			// code that is repeated every cycle in this state	
				IF iCurrentValveMode = 63 AND iCurrentChannelTM = 31 AND iCurrentTransferControlTM = 2 AND iCurrentAddressedTargetTM = usiChooseOtherValve AND iCurrentIndexTM = iCountMFLdownload + 50 THEN
					astMalfunctionlist[iCountMFLdownload].uiHours := WORD_TO_UINT(awBusDataFromVTEM[2]);				// Save hours
					
					xStateFinished := TRUE;
				END_IF
			//-----------------------------------------------------------------------------------------------------------
			
			// Transition
				IF xStateFinished = TRUE THEN
					xStateFinished := FALSE;
					xStateChange := TRUE;
					iState := 42;
					iCommandNumber := 42;
				END_IF
			//-----------------------------------------------------------------------------------------------------------
			
		42:	// READING MALFUNCTION MESSAGE TIME STAMP PART II
			// code that is executed only in the first cycle of this state
				IF xStateChange = TRUE THEN
					xStateChange := FALSE;
					iResponse := eResponseReadMalfunctionList.transferring;
					xDone := FALSE;
					xError := FALSE;
					xBusy := TRUE;
					xAborted := FALSE;
				END_IF
			//-----------------------------------------------------------------------------------------------------------

			// code that is repeated every cycle in this state	
				IF iCurrentValveMode = 63 AND iCurrentChannelTM = 31 AND iCurrentTransferControlTM = 2 AND iCurrentAddressedTargetTM = usiChooseOtherValve AND iCurrentIndexTM = iCountMFLdownload + 100 THEN
					fbreadbitsfromword(wData:=awBusDataFromVTEM[2], iStartBit:=8, iEndBit:=15, iValue:= , xError:=);		// Read minutes
					astMalfunctionlist[iCountMFLdownload].usiMinutes := INT_TO_USINT(fbreadbitsfromword.iValue);			// Save minutes
					
					fbreadbitsfromword(wData:=awBusDataFromVTEM[2], iStartBit:=0, iEndBit:=7, iValue:= , xError:=);			// Read seconds
					astMalfunctionlist[iCountMFLdownload].usiSeconds := INT_TO_USINT(fbreadbitsfromword.iValue);			// Save seconds
					
					xStateFinished := TRUE;
				END_IF
			//-----------------------------------------------------------------------------------------------------------
			
			// Transition
				IF xStateFinished = TRUE THEN
					xStateFinished := FALSE;
					xStateChange := TRUE;
					iState := 43;
					iCommandNumber := 43;
				END_IF
			//-----------------------------------------------------------------------------------------------------------

		43:	// READING MALFUNCTION MESSAGE TIME STAMP PART III
			// code that is executed only in the first cycle of this state
				IF xStateChange = TRUE THEN
					xStateChange := FALSE;
					iResponse := eResponseReadMalfunctionList.transferring;
					xDone := FALSE;
					xError := FALSE;
					xBusy := TRUE;
					xAborted := FALSE;
				END_IF
			//-----------------------------------------------------------------------------------------------------------
			
			// code that is repeated every cycle in this state	
				IF iCurrentValveMode = 63 AND iCurrentChannelTM = 31 AND iCurrentTransferControlTM = 2 AND iCurrentAddressedTargetTM = usiChooseOtherValve AND iCurrentIndexTM = iCountMFLdownload + 150 THEN
					astMalfunctionlist[iCountMFLdownload].uiMilliseconds := WORD_TO_UINT(awBusDataFromVTEM[2]);			// Save milliseconds
					
					IF iCountMFLdownload = iNumberOfMalfunctions THEN
						xReadProcessFinished := TRUE;
					ELSE
						xReadProcessFinished := FALSE;
						xStateFinished := TRUE;
					END_IF
				END_IF
			//-----------------------------------------------------------------------------------------------------------
			
			// Transition
				IF xReadProcessFinished = TRUE THEN
					xStateChange := TRUE;
					xStateFinished := FALSE;
					iState := 44;
					iCommandNumber := 44;
				ELSIF xStateFinished = TRUE THEN
					xStateFinished := FALSE;
					xStateChange := TRUE;
					iState := 40;
					iCountMFLdownload := iCountMFLdownload + 1;
					iCommandNumber := 40;
				END_IF
			//-----------------------------------------------------------------------------------------------------------
			
		44:	// READING TIME CODE OF MALFUNCTION LIST PART I
			// code that is executed only in the first cycle of this state
				IF xStateChange = TRUE THEN
					xStateChange := FALSE;
					iResponse := eResponseReadMalfunctionList.transferring;
					xDone := FALSE;
					xError := FALSE;
					xBusy := TRUE;
					xAborted := FALSE;
				END_IF
			//-----------------------------------------------------------------------------------------------------------
			
			// code that is repeated every cycle in this state	
				IF iCurrentValveMode = 63 AND iCurrentChannelTM = 31 AND iCurrentTransferControlTM = 2 AND iCurrentAddressedTargetTM = usiChooseOtherValve AND iCurrentIndexTM = 250 THEN
					stTimeStampList.uiHours := WORD_TO_UINT(awBusDataFromVTEM[2]);											// Save Hours
					
					xStateFinished := TRUE;
				END_IF
			//-----------------------------------------------------------------------------------------------------------
			
			// Transition
				IF xStateFinished = TRUE THEN
					xStateFinished := FALSE;
					xStateChange := TRUE;
					iState := 45;
					iCommandNumber := 45;
				END_IF
			//-----------------------------------------------------------------------------------------------------------
		
		45:	// READING TIME CODE OF MALFUNCTION LIST PART III
			// code that is executed only in the first cycle of this state
				IF xStateChange = TRUE THEN
					xStateChange := FALSE;
					iResponse := eResponseReadMalfunctionList.transferring;
					xDone := FALSE;
					xError := FALSE;
					xBusy := TRUE;
					xAborted := FALSE;
				END_IF
			//-----------------------------------------------------------------------------------------------------------
			
			// code that is repeated every cycle in this state	
				IF iCurrentValveMode = 63 AND iCurrentChannelTM = 31 AND iCurrentTransferControlTM = 2 AND iCurrentAddressedTargetTM = usiChooseOtherValve AND iCurrentIndexTM = 251 THEN
					fbreadbitsfromword(wData:=awBusDataFromVTEM[2], iStartBit:=8, iEndBit:=15, iValue:= , xError:=);		// Read minutes
					stTimeStampList.usiMinutes := INT_TO_USINT(fbreadbitsfromword.iValue);									// Save minutes

					fbreadbitsfromword(wData:=awBusDataFromVTEM[2], iStartBit:=0, iEndBit:=7, iValue:= , xError:=);			// Read seconds
					stTimeStampList.usiSeconds := INT_TO_USINT(fbreadbitsfromword.iValue);									// Save seconds
					
					xStateFinished := TRUE;
				END_IF
			//-----------------------------------------------------------------------------------------------------------
			
			// Transition
				IF xStateFinished = TRUE THEN
					xStateFinished := FALSE;
					xStateChange := TRUE;
					iState := 46;
					iCommandNumber := 46;
				END_IF
			//-----------------------------------------------------------------------------------------------------------
		
		46:	// READING TIME CODE OF MALFUNCTION LIST PART III
			// code that is executed only in the first cycle of this state
				IF xStateChange = TRUE THEN
					xStateChange := FALSE;
					iResponse := eResponseReadMalfunctionList.transferring;
					xDone := FALSE;
					xError := FALSE;
					xBusy := TRUE;
					xAborted := FALSE;
				END_IF
			//-----------------------------------------------------------------------------------------------------------
			
			// code that is repeated every cycle in this state	
				IF iCurrentValveMode = 63 AND iCurrentChannelTM = 31 AND iCurrentTransferControlTM = 2 AND iCurrentAddressedTargetTM = usiChooseOtherValve AND iCurrentIndexTM = 252 THEN
					stTimeStampList.uiMilliseconds := WORD_TO_UINT(awBusDataFromVTEM[2]);									// Save milliseconds
					
					xStateFinished := TRUE;
				END_IF
			//-----------------------------------------------------------------------------------------------------------
			
			// Transition
				IF xStateFinished = TRUE THEN
					xStateFinished := FALSE;
					xStateChange := TRUE;
					iState := 50;
				END_IF
			//-----------------------------------------------------------------------------------------------------------
		
		50:	// DONE
			// code that is executed only in the first cycle of this state
				IF xStateChange = TRUE THEN
					xStateChange := FALSE;
					iResponse := eResponseReadMalfunctionList.done;
					xDone := TRUE;
					xError := FALSE;
					xBusy := FALSE;
					xAborted := FALSE;
				END_IF
			//-----------------------------------------------------------------------------------------------------------
			
			// code that is repeated every cycle in this state	
				iCommandNumber := 5;	// exit transfer mode
			//-----------------------------------------------------------------------------------------------------------
			
			// Transition
				IF xExecute = FALSE THEN
					xStateChange := TRUE;
					iState := 100;
				END_IF
			//-----------------------------------------------------------------------------------------------------------
			
		51:	// DONE WITH EMPTY MALFUNCTION LIST
			// code that is executed only in the first cycle of this state
				IF xStateChange = TRUE THEN
					xStateChange := FALSE;
					iResponse := eResponseReadMalfunctionList.no_entries_in_malfunction_list;
					xDone := TRUE;
					xError := FALSE;
					xBusy := FALSE;
					xAborted := FALSE;
				END_IF
			//-----------------------------------------------------------------------------------------------------------
			
			// code that is repeated every cycle in this state	
				iCommandNumber := 5;	// exit transfer mode
			//-----------------------------------------------------------------------------------------------------------
			
			// Transition
				IF xExecute = FALSE THEN
					xStateChange := TRUE;
					iState := 100;
				END_IF
			//-----------------------------------------------------------------------------------------------------------
			
		70:	// ERROR
			// code that is executed only in the first cycle of this state
				IF xStateChange = TRUE THEN
					xStateChange := FALSE;
					iResponse := eResponseReadMalfunctionList.error_while_transmitting_data_to_vtem;
					xDone := FALSE;
					xError := TRUE;
					xBusy := FALSE;
					xAborted := FALSE;
				END_IF
			//-----------------------------------------------------------------------------------------------------------
				IF xInputConsistent = FALSE THEN
					iResponse := eResponseReadMalfunctionList.FB_needs_rising_edge_xExecute;
				END_IF
			
			// code that is repeated every cycle in this state	
				CASE iCurrentAppState OF
					1:	iResponse := eResponseReadMalfunctionList.invalid_SetValveMode;
					2:	iResponse := eResponseReadMalfunctionList.invalid_SetAppControl;
					3:	iResponse := eResponseReadMalfunctionList.invalid_SetAppOption;
					4:	iResponse := eResponseReadMalfunctionList.invalid_SetPointValue1;
					5:	iResponse := eResponseReadMalfunctionList.invalid_SetPointValue2;
					6:	iResponse := eResponseReadMalfunctionList.invalid_configuration;
					
					10:	iResponse := eResponseReadMalfunctionList.access_denied_WebConfig;
					11:	iResponse := eResponseReadMalfunctionList.access_denied_saving_parameterisation;
					12:	iResponse := eResponseReadMalfunctionList.no_license_for_this_MA;
					13:	iResponse := eResponseReadMalfunctionList.all_licenses_in_use;
					14:	iResponse := eResponseReadMalfunctionList.invalid_license_file;
					15:	iResponse := eResponseReadMalfunctionList.no_valve_detected;
					16:	iResponse := eResponseReadMalfunctionList.valve_self_calibration_running;
				END_CASE
			//-----------------------------------------------------------------------------------------------------------
			
			// Transition
				IF xExecute = FALSE AND xAbort = FALSE THEN
					xStateChange := TRUE;
					iState := 100;
				END_IF
			//-----------------------------------------------------------------------------------------------------------
			
		71:	// ERROR DURING TRANFER MODE
			// code that is executed only in the first cycle of this state
				IF xStateChange = TRUE THEN
					xStateChange := FALSE;
					xDone := FALSE;
					xError := TRUE;
					xBusy := FALSE;
					xAborted := FALSE;
				END_IF
			//-----------------------------------------------------------------------------------------------------------
			
			// code that is repeated every cycle in this state	
				CASE iCurrentValueTM OF
					1:	iResponse := eResponseReadMalfunctionList.invalid_Channel;
					2:	iResponse := eResponseReadMalfunctionList.invalid_TransferControl;
					3:	iResponse := eResponseReadMalfunctionList.invalid_usiChooseOtherValve; // invalid_AddtessedTarget is always invalid_usiChooseOtherValve
					4:	iResponse := eResponseReadMalfunctionList.invalid_Index;
					5:	iResponse := eResponseReadMalfunctionList.invalid_TransferValue;
					6:	iResponse := eResponseReadMalfunctionList.no_data_empty_slot;	// invalid_Combination is always no_data_empty_slot in the context of this function block
					7:	iResponse := eResponseReadMalfunctionList.access_denied_DataInUse;
					8:	iResponse := eResponseReadMalfunctionList.no_data_empty_slot;
				END_CASE
			//-----------------------------------------------------------------------------------------------------------
			
			// Transition
				IF xExecute = FALSE AND xAbort = FALSE THEN
					xStateChange := TRUE;
					iState := 100;
				END_IF
			//-----------------------------------------------------------------------------------------------------------
			
		80:	// ABORTING
			// code that is executed only in the first cycle of this state
				IF xStateChange = TRUE THEN
					xStateChange := FALSE;
					iResponse := eResponseReadMalfunctionList.aborting;
					xBusy := FALSE;
					xDone := FALSE;
					xError := FALSE;
					xAborted := TRUE;
				END_IF
			//-----------------------------------------------------------------------------------------------------------
			
			// code that is repeated every cycle in this state
				IF iCurrentValveMode = 63 THEN
					iCommandNumber := 5;	// exit transfer mode
				ELSIF iCurrentValveMode <> 61 AND iCurrentValveMode <> 63 THEN
					iCommandNumber := 6;	// stop running motion apps
				ELSE
					iCommandNumber := 0; 
				END_IF
			//-----------------------------------------------------------------------------------------------------------
			
			// Transition
				IF xAbort = FALSE AND xExecute = FALSE AND iCurrentValveMode = 61 THEN
					xStateChange := TRUE;
					iState := 100;
				END_IF
			//-----------------------------------------------------------------------------------------------------------

		100:	// RESETTING FUNCTION BLOCK AND VALVE
			// code that is executed only in the first cycle of this state
				IF xStateChange = TRUE THEN
					xStateChange := FALSE;
					iResponse := eResponseReadMalfunctionList.resetting;
					xDone := FALSE;
					xError := FALSE;
					xBusy := FALSE;
					xAborted := FALSE;
					xFirstTransfer := FALSE;
				END_IF
			//-----------------------------------------------------------------------------------------------------------
			
			// code that is repeated every cycle in this state	
				IF iCurrentValveMode = 63 THEN
					iCommandNumber := 5;	// exit transfer mode
				ELSIF iCurrentValveMode <> 61 AND iCurrentValveMode <> 63 THEN
					iCommandNumber := 6;	// stop running motion apps
				END_IF
				
				FOR iCountMFLreset := 1 TO 40 BY 1 DO
					astMalfunctionlist[iCountMFLreset].usiMalfunctionCode := 0;
					astMalfunctionlist[iCountMFLreset].usiMalfunctionSubcode := 0;
					astMalfunctionlist[iCountMFLreset].usiMalfunctionClassification := 0;
					astMalfunctionlist[iCountMFLreset].uiHours := 0;
					astMalfunctionlist[iCountMFLreset].usiMinutes := 0;
					astMalfunctionlist[iCountMFLreset].usiSeconds := 0;
					astMalfunctionlist[iCountMFLreset].uiMilliseconds := 0;
				END_FOR
				
				stTimeStampList.uiHours := 0;
				stTimeStampList.usiMinutes := 0;
				stTimeStampList.usiSeconds := 0;
				stTimeStampList.uiMilliseconds := 0;
				
				iNumberOfMalfunctions := 0;
				
				iCountMFLreset := 0;
				iCountMFLdownload := 1;
				xReadProcessFinished := FALSE;
				xStateFinished := FALSE;
			//-----------------------------------------------------------------------------------------------------------
			
			// Transition
				IF iCurrentValveMode = 61 THEN
					iCommandNumber := 6; // Last command to send before the FB is in IDLE
					xStateChange := TRUE;
					iState := 10;
				END_IF
			//-----------------------------------------------------------------------------------------------------------
			
	END_CASE
//-----------------------------------------------------------------------------------------------------------

// command section
	CASE iCommandNumber OF
		0:	// IDLE
			;
		
		5:	// EXIT TRANSFER MODE
			fbwritevaluetoword(iValue:=63, iStartBit:=0, iEndBit:=5, wDataWord:=awBusDataToVTEM[0], xError=> );							// Valve Mode = 63
			fbwritevaluetoword(iValue:=0, iStartBit:=6, iEndBit:=7, wDataWord:=awBusDataToVTEM[0], xError=> );							// 0 (unused)
			fbwritevaluetoword(iValue:=0, iStartBit:=8, iEndBit:=12, wDataWord:=awBusDataToVTEM[0], xError=> );							// Channel = 0 (ignored)
			fbwritevaluetoword(iValue:=3, iStartBit:=13, iEndBit:=15, wDataWord:=awBusDataToVTEM[0], xError=> );						// Transfer Control = Exit transfer mode (3)
			fbwritevaluetoword(iValue:=0, iStartBit:=0, iEndBit:=7, wDataWord:=awBusDataToVTEM[1], xError=> );							// Addressed Target = 0 (ignored)
			fbwritevaluetoword(iValue:=0, iStartBit:=8, iEndBit:=15, wDataWord:=awBusDataToVTEM[1], xError=> );							// Index = 0 (ignored)
			fbwritevaluetoword(iValue:=0, iStartBit:=0, iEndBit:=15, wDataWord:=awBusDataToVTEM[2], xError=> );							// Value = 0 (ignored)
			
		6:	// stop running motion apps
			fbwritevaluetoword(iValue:=61, iStartBit:=0, iEndBit:=5, wDataWord:=awBusDataToVTEM[0], xError=> );							// Valve Mode = 61 (stop)
			fbwritevaluetoword(iValue:=0, iStartBit:=6, iEndBit:=7, wDataWord:=awBusDataToVTEM[0], xError=> );							// App Control = 0 (unused)
			fbwritevaluetoword(iValue:=0, iStartBit:=8, iEndBit:=15, wDataWord:=awBusDataToVTEM[0], xError=> );							// App Option = 0 (unused)
			fbwritevaluetoword(iValue:=0, iStartBit:=0, iEndBit:=15, wDataWord:=awBusDataToVTEM[1], xError=> );							// Setpoint Value 1 = 0 (unused)
			fbwritevaluetoword(iValue:=0, iStartBit:=0, iEndBit:=15, wDataWord:=awBusDataToVTEM[2], xError=> );							// Setpoint Value 2 = 0 (unused)
		
		10:	// getting count of malfunction messages
			fbwritevaluetoword(iValue:=63, iStartBit:=0, iEndBit:=5, wDataWord:=awBusDataToVTEM[0], xError=> );							// Valve Mode = 63 (transfer mode)
			fbwritevaluetoword(iValue:=0, iStartBit:=6, iEndBit:=7, wDataWord:=awBusDataToVTEM[0], xError=> );							// 0 (unused)
			fbwritevaluetoword(iValue:=31, iStartBit:=8, iEndBit:=12, wDataWord:=awBusDataToVTEM[0], xError=> );						// Channel = 31 (malfunctions)
			fbwritevaluetoword(iValue:=2, iStartBit:=13, iEndBit:=15, wDataWord:=awBusDataToVTEM[0], xError=> );						// Transfer Control = 2 (Upload)
			fbwritevaluetoword(iValue:=usiChooseOtherValve, iStartBit:=0, iEndBit:=7, wDataWord:=awBusDataToVTEM[1], xError=> );		// Addressed Target = usiChooseOtherValve
			fbwritevaluetoword(iValue:=255, iStartBit:=8, iEndBit:=15, wDataWord:=awBusDataToVTEM[1], xError=> );						// Index = 255 (Number of malfunction messages)
			fbwritevaluetoword(iValue:=0, iStartBit:=0, iEndBit:=15, wDataWord:=awBusDataToVTEM[2], xError=> );							// Value = 0 (Upload)
		
		40:	// reading malfunction list
			fbwritevaluetoword(iValue:=63, iStartBit:=0, iEndBit:=5, wDataWord:=awBusDataToVTEM[0], xError=> );							// Valve Mode = 63 (transfer mode)
			fbwritevaluetoword(iValue:=0, iStartBit:=6, iEndBit:=7, wDataWord:=awBusDataToVTEM[0], xError=> );							// 0 (unused)
			fbwritevaluetoword(iValue:=31, iStartBit:=8, iEndBit:=12, wDataWord:=awBusDataToVTEM[0], xError=> );						// Channel = 31 (malfunctions)
			fbwritevaluetoword(iValue:=2, iStartBit:=13, iEndBit:=15, wDataWord:=awBusDataToVTEM[0], xError=> );						// Transfer Control = 2 (Upload)
			fbwritevaluetoword(iValue:=usiChooseOtherValve, iStartBit:=0, iEndBit:=7, wDataWord:=awBusDataToVTEM[1], xError=> );		// Addressed Target = usiChooseOtherValve
			fbwritevaluetoword(iValue:=iCountMFLdownload, iStartBit:=8, iEndBit:=15, wDataWord:=awBusDataToVTEM[1], xError=> );			// Index = iCounterMFLdownload (malfunction message)
			fbwritevaluetoword(iValue:=0, iStartBit:=0, iEndBit:=15, wDataWord:=awBusDataToVTEM[2], xError=> );							// Value = 0 (Upload)

		41:	// reading malfunction entry time stamp part I
			fbwritevaluetoword(iValue:=63, iStartBit:=0, iEndBit:=5, wDataWord:=awBusDataToVTEM[0], xError=> );							// Valve Mode = 63 (transfer mode)
			fbwritevaluetoword(iValue:=0, iStartBit:=6, iEndBit:=7, wDataWord:=awBusDataToVTEM[0], xError=> );							// 0 (unused)
			fbwritevaluetoword(iValue:=31, iStartBit:=8, iEndBit:=12, wDataWord:=awBusDataToVTEM[0], xError=> );						// Channel = 31 (malfunctions)
			fbwritevaluetoword(iValue:=2, iStartBit:=13, iEndBit:=15, wDataWord:=awBusDataToVTEM[0], xError=> );						// Transfer Control = 2 (Upload)
			fbwritevaluetoword(iValue:=usiChooseOtherValve, iStartBit:=0, iEndBit:=7, wDataWord:=awBusDataToVTEM[1], xError=> );		// Addressed Target = usiChooseOtherValve
			fbwritevaluetoword(iValue:=iCountMFLdownload+50, iStartBit:=8, iEndBit:=15, wDataWord:=awBusDataToVTEM[1], xError=> );		// Index = iCounterMFLdownload + 50 (time stamp of malfunction message, part I)
			fbwritevaluetoword(iValue:=0, iStartBit:=0, iEndBit:=15, wDataWord:=awBusDataToVTEM[2], xError=> );							// Value = 0 (Upload)
			
		42:	// reading malfunction entry time stamp part II
			fbwritevaluetoword(iValue:=63, iStartBit:=0, iEndBit:=5, wDataWord:=awBusDataToVTEM[0], xError=> );							// Valve Mode = 63 (transfer mode)
			fbwritevaluetoword(iValue:=0, iStartBit:=6, iEndBit:=7, wDataWord:=awBusDataToVTEM[0], xError=> );							// 0 (unused)
			fbwritevaluetoword(iValue:=31, iStartBit:=8, iEndBit:=12, wDataWord:=awBusDataToVTEM[0], xError=> );						// Channel = 31 (malfunctions)
			fbwritevaluetoword(iValue:=2, iStartBit:=13, iEndBit:=15, wDataWord:=awBusDataToVTEM[0], xError=> );						// Transfer Control = 2 (Upload)
			fbwritevaluetoword(iValue:=usiChooseOtherValve, iStartBit:=0, iEndBit:=7, wDataWord:=awBusDataToVTEM[1], xError=> );		// Addressed Target = usiChooseOtherValve
			fbwritevaluetoword(iValue:=iCountMFLdownload+100, iStartBit:=8, iEndBit:=15, wDataWord:=awBusDataToVTEM[1], xError=> );		// Index = iCounterMFLdownload + 100 (time stamp of malfunction message, part II)
			fbwritevaluetoword(iValue:=0, iStartBit:=0, iEndBit:=15, wDataWord:=awBusDataToVTEM[2], xError=> );							// Value = 0 (Upload)

		43: // reading malfunction entry time stamp part III
			fbwritevaluetoword(iValue:=63, iStartBit:=0, iEndBit:=5, wDataWord:=awBusDataToVTEM[0], xError=> );							// Valve Mode = 63 (transfer mode)
			fbwritevaluetoword(iValue:=0, iStartBit:=6, iEndBit:=7, wDataWord:=awBusDataToVTEM[0], xError=> );							// 0 (unused)
			fbwritevaluetoword(iValue:=31, iStartBit:=8, iEndBit:=12, wDataWord:=awBusDataToVTEM[0], xError=> );						// Channel = 31 (malfunctions)
			fbwritevaluetoword(iValue:=2, iStartBit:=13, iEndBit:=15, wDataWord:=awBusDataToVTEM[0], xError=> );						// Transfer Control = 2 (Upload)
			fbwritevaluetoword(iValue:=usiChooseOtherValve, iStartBit:=0, iEndBit:=7, wDataWord:=awBusDataToVTEM[1], xError=> );		// Addressed Target = usiChooseOtherValve
			fbwritevaluetoword(iValue:=iCountMFLdownload+150, iStartBit:=8, iEndBit:=15, wDataWord:=awBusDataToVTEM[1], xError=> );		// Index = iCounterMFLdownload + 150 (time stamp of malfunction message, part III)
			fbwritevaluetoword(iValue:=0, iStartBit:=0, iEndBit:=15, wDataWord:=awBusDataToVTEM[2], xError=> );							// Value = 0 (Upload)
		
		44:	// reading time stamp of malfunction list part I
			fbwritevaluetoword(iValue:=63, iStartBit:=0, iEndBit:=5, wDataWord:=awBusDataToVTEM[0], xError=> );							// Valve Mode = 63 (transfer mode)
			fbwritevaluetoword(iValue:=0, iStartBit:=6, iEndBit:=7, wDataWord:=awBusDataToVTEM[0], xError=> );							// 0 (unused)
			fbwritevaluetoword(iValue:=31, iStartBit:=8, iEndBit:=12, wDataWord:=awBusDataToVTEM[0], xError=> );						// Channel = 31 (malfunctions)
			fbwritevaluetoword(iValue:=2, iStartBit:=13, iEndBit:=15, wDataWord:=awBusDataToVTEM[0], xError=> );						// Transfer Control = 2 (Upload)
			fbwritevaluetoword(iValue:=usiChooseOtherValve, iStartBit:=0, iEndBit:=7, wDataWord:=awBusDataToVTEM[1], xError=> );		// Addressed Target = usiChooseOtherValve
			fbwritevaluetoword(iValue:=250, iStartBit:=8, iEndBit:=15, wDataWord:=awBusDataToVTEM[1], xError=> );						// Index = 250 (time stamp of malfunction list, part I)
			fbwritevaluetoword(iValue:=0, iStartBit:=0, iEndBit:=15, wDataWord:=awBusDataToVTEM[2], xError=> );							// Value = 0 (Upload)
		
		45:	// reading time stamp of malfunction list part II
			fbwritevaluetoword(iValue:=63, iStartBit:=0, iEndBit:=5, wDataWord:=awBusDataToVTEM[0], xError=> );							// Valve Mode = 63 (transfer mode)
			fbwritevaluetoword(iValue:=0, iStartBit:=6, iEndBit:=7, wDataWord:=awBusDataToVTEM[0], xError=> );							// 0 (unused)
			fbwritevaluetoword(iValue:=31, iStartBit:=8, iEndBit:=12, wDataWord:=awBusDataToVTEM[0], xError=> );						// Channel = 31 (malfunctions)
			fbwritevaluetoword(iValue:=2, iStartBit:=13, iEndBit:=15, wDataWord:=awBusDataToVTEM[0], xError=> );						// Transfer Control = 2 (Upload)
			fbwritevaluetoword(iValue:=usiChooseOtherValve, iStartBit:=0, iEndBit:=7, wDataWord:=awBusDataToVTEM[1], xError=> );		// Addressed Target = usiChooseOtherValve
			fbwritevaluetoword(iValue:=251, iStartBit:=8, iEndBit:=15, wDataWord:=awBusDataToVTEM[1], xError=> );						// Index = 251 (time stamp of malfunction list, part II)
			fbwritevaluetoword(iValue:=0, iStartBit:=0, iEndBit:=15, wDataWord:=awBusDataToVTEM[2], xError=> );							// Value = 0 (Upload)
		
		46:	// reading time stamp of malfunction list part III
			fbwritevaluetoword(iValue:=63, iStartBit:=0, iEndBit:=5, wDataWord:=awBusDataToVTEM[0], xError=> );							// Valve Mode = 63 (transfer mode)
			fbwritevaluetoword(iValue:=0, iStartBit:=6, iEndBit:=7, wDataWord:=awBusDataToVTEM[0], xError=> );							// 0 (unused)
			fbwritevaluetoword(iValue:=31, iStartBit:=8, iEndBit:=12, wDataWord:=awBusDataToVTEM[0], xError=> );						// Channel = 31 (malfunctions)
			fbwritevaluetoword(iValue:=2, iStartBit:=13, iEndBit:=15, wDataWord:=awBusDataToVTEM[0], xError=> );						// Transfer Control = 2 (Upload)
			fbwritevaluetoword(iValue:=usiChooseOtherValve, iStartBit:=0, iEndBit:=7, wDataWord:=awBusDataToVTEM[1], xError=> );		// Addressed Target = usiChooseOtherValve
			fbwritevaluetoword(iValue:=252, iStartBit:=8, iEndBit:=15, wDataWord:=awBusDataToVTEM[1], xError=> );						// Index = 252 (time stamp of malfunction list, part III)
			fbwritevaluetoword(iValue:=0, iStartBit:=0, iEndBit:=15, wDataWord:=awBusDataToVTEM[2], xError=> );							// Value = 0 (Upload)

	END_CASE	
//-----------------------------------------------------------------------------------------------------------

END_FUNCTION_BLOCK

// Transfermode/specific_MA_config/FB_Write_config_MA_10
// This function block can be used to download the configuration of Motion App 10 ("Flow control").
// The specific parameters of this Motion App are the inputs of this FB and can be defined by the user. 
// The function block uses the transfer mode to write this configuration to the Motion Terminal
// and indicates the state of the download process.

FUNCTION_BLOCK FB_Write_config_MA_10
VAR_INPUT
	awBusDataFromVTEM 				: ARRAY [0..2] OF WORD;		(* 6 bytes of process data received from the Motion Terminal *)
END_VAR
	
VAR_IN_OUT
	awBusDataToVTEM 				: ARRAY [0..2] OF WORD; 	(* 6 bytes of process data sent to the Motion Terminal *)
END_VAR

VAR_INPUT
	xExecute 						: BOOL; 					(* has to be set to TRUE for a download and to FALSE to reset the function block after a download *)

	iParameterSet					: INT := 1; 				(* the parameter set to be written to, 1 by default *)
	
	// system parameters
		iOperatingMedium			: eMA10OperatingMedium := 1;// Type and condition of the operating medium (values see eMA10OperatingMedium)
		iInPortFlowRate2_optional	: INT;						// Sensor port for flow rate at (2) (required for closed-loop controlled operating mode, value is number of the slot (beginning from 0 and including valve slots) * 10 + number of the port 
		iInPortFlowRate4_optional	: INT;						// Sensor port for flow rate at (4) (required for closed-loop controlled operating mode, value is number of the slot (beginning from 0 and including valve slots) * 10 + number of the port
		iInPortRetracted_optional	: INT;						// Sensor port for detection of end position at pressurisation of outlet port 2 (retracted), value is number of the slot (beginning from 0 and including valve slots) * 10 + number of the port
		iInPortAdvanced_optional	: INT;						// Sensor port for detection of end position at pressurisation of outlet port 4 (advanced), value is number of the slot (beginning from 0 and including valve slots) * 10 + number of the port

	// application parameters
		iCharacteristicAt2			: INT;						// Control characteristic, outlet port (2) (0 = "fast" (short tubes), 1 = medium (medium length tubes), 2 = "universal" (esp. long tubes), 3 = defined by tuning parameters (only if closed-loop control is activated for outlet port (2)))
		iCharacteristicAt4			: INT;						// Control characteristic, outlet port (4) (0 = "fast" (short tubes), 1 = medium (medium length tubes), 2 = "universal" (esp. long tubes), 3 = defined by tuning parameters (only if closed-loop control is activated for outlet port (4)))
		xClosedLoopControl2			: BOOL := FALSE;			// TRUE acivates closed-loop control for outlet port (2), FALSE is open-loop controlled operation
		xClosedLoopControl4			: BOOL := FALSE;			// TRUE acivates closed-loop control for outlet port (4), FALSE is open-loop controlled operation
		
	// tuning parameters
		iOptProportionalGainFor2	: INT;						// Optional tuning parameter for the customized proportional element of the PID modulator at outlet port (2) [1 digit = 0.01 g/s/bar]
		iOptIntegralGainFor2		: INT;						// Optional tuning parameter for the customized integral element of the PID modulator at outlet port (2) [1 digit = 0.01 g/s²/bar]
		iOptRedFeedforwContrRate2	: INT;						// Optional tuning parameter for reduction of feedforward control rate of 100% for outlet port (2) [1 digit = 1%]
		iOptBoostSetpointReach2		: INT;						// Optional tuning parameter for boost to reach the setpoint value for outlet port (2) earlier, but with higher overshoot [1 digit = 1%] 
		iOptOffsetTargFRLimitInfo2	: INT;						// Optional tuning parameter for offset on the threshold value of 95% of the possible relative flow at outlet port (2) for feedback in app state, bit 5 [1 digit = 1%]
		iOptOffsetMinConsSetp2		: INT;						// Optional tuning parameter for offset to the threshold value of 25 l/min, below which a target flow rate for outlet port (2) is not considered [1 digit = 1 l/min]

		iOptProportionalGainFor4	: INT;						// Optional tuning parameter for the customized proportional element of the PID modulator at outlet port (4) [1 digit = 0.01 g/s/bar]
		iOptIntegralGainFor4		: INT;						// Optional tuning parameter for the customized integral element of the PID modulator at outlet port (4) [1 digit = 0.01 g/s²/bar]
		iOptRedFeedforwContrRate4	: INT;						// Optional tuning parameter for reduction of feedforward control rate of 100% for outlet port (4) [1 digit = 1%]
		iOptBoostSetpointReach4		: INT;						// Optional tuning parameter for boost to reach the setpoint value for outlet port (4) earlier, but with higher overshoot [1 digit = 1%] 
		iOptOffsetTargFRLimitInfo4	: INT;						// Optional tuning parameter for offset on the threshold value of 95% of the possible relative flow at outlet port (4) for feedback in app state, bit 5 [1 digit = 1%]
		iOptOffsetMinConsSetp4		: INT;						// Optional tuning parameter for offset to the threshold value of 25 l/min, below which a target flow rate for outlet port (4) is not considered [1 digit = 1 l/min]
END_VAR

VAR_OUTPUT                  		
	iResponse 						: eTransferResponse; 		(* returns the status of the execution of the download process *)
	sCurrentValue 					: STRING; 					(* indicates which value of the array is currently treated (necessary to evaluate in case of error messages) *)
	xDownloadDone 					: BOOL; 					(* indicates whether the download was successful *)
	xDownloadError 					: BOOL := FALSE; 			(* indicates whether an error occurred during the transfer *)
END_VAR

VAR
	aTransferPackages				: ARRAY [0..100] OF stTransferPackage;
	fbdownloadMultipleParameters 	: FB_Download_Multiple_Parameters;
	iCurrentValue					: INT;
	fbWriteValueToWord 				: FB_Write_Value_To_Word;
	iOperatingMode					: INT;						// Container for the information of the variables xClosedLoopControl2 and xClosedLoopControl4
	wOperatingMode					: WORD;						// word container for the operating mode
END_VAR

(*****************************************************************************************************

Festo SE & Co. KG, Esslingen
Copyright (c) 2020. All rights reserved.

Product:            Motion Terminal VTEM
Description:        Function Block to download the parameters for Motion App 10 to the Motion Terminal

Object version:     1.00
Last change:        2021-02
======================================================================================================
                                       H I S T O R Y
======================================================================================================
Version:            1.00
Date:               2021-02
Change/Activity:    - created (#3805775)
Release:            3.5.7.236 (CODESYS 3.5.7.2, Lib version 3.6)
Author:             JEBU
======================================================================================================

*****************************************************************************************************)

// combine xClosedLoopControl2 and xClosedLoopControl4 into iOperatingMode (Bit 0 = (4), Bit 1 = (2))
	wOperatingMode.0 := xClosedLoopControl4;
	wOperatingMode.1 := xClosedLoopControl2; 
	iOperatingMode := WORD_TO_INT(wOperatingMode);

// write the Motion App specific parameters into the struct
	//iOperatingMedium
		aTransferPackages[0].iChannel := iParameterSet;
		aTransferPackages[0].iAddressedTarget := 10;
		aTransferPackages[0].iIndex := 42;
		aTransferPackages[0].iTransferValue := iOperatingMedium;
	
	//iInPortFlowRate2_optional
		aTransferPackages[1].iChannel := iParameterSet;
		aTransferPackages[1].iAddressedTarget := 10;
		aTransferPackages[1].iIndex := 81;
		aTransferPackages[1].iTransferValue := iInPortFlowRate2_optional;

	//iInPortFlowRate4_optional
		aTransferPackages[2].iChannel := iParameterSet;
		aTransferPackages[2].iAddressedTarget := 10;
		aTransferPackages[2].iIndex := 82;
		aTransferPackages[2].iTransferValue := iInPortFlowRate4_optional;
	
	//iInPortRetracted_optional
		aTransferPackages[3].iChannel := iParameterSet;
		aTransferPackages[3].iAddressedTarget := 10;
		aTransferPackages[3].iIndex := 70;
		aTransferPackages[3].iTransferValue := iInPortRetracted_optional;
	
	//iInPortAdvanced_optional
		aTransferPackages[4].iChannel := iParameterSet;
		aTransferPackages[4].iAddressedTarget := 10;
		aTransferPackages[4].iIndex := 71;
		aTransferPackages[4].iTransferValue := iInPortAdvanced_optional;
	
	//iCharacteristicAt2
		aTransferPackages[5].iChannel := iParameterSet;
		aTransferPackages[5].iAddressedTarget := 10;
		aTransferPackages[5].iIndex := 220;
		aTransferPackages[5].iTransferValue := iCharacteristicAt2;
	
	//iCharacteristicAt4
		aTransferPackages[6].iChannel := iParameterSet;
		aTransferPackages[6].iAddressedTarget := 10;
		aTransferPackages[6].iIndex := 221;
		aTransferPackages[6].iTransferValue := iCharacteristicAt4;
	
	//iOperatingMode
		aTransferPackages[7].iChannel := iParameterSet;
		aTransferPackages[7].iAddressedTarget := 10;
		aTransferPackages[7].iIndex := 223;
		aTransferPackages[7].iTransferValue := iOperatingMode;
	
	//iOptProportionalGainFor2
		aTransferPackages[8].iChannel := iParameterSet;
		aTransferPackages[8].iAddressedTarget := 10;
		aTransferPackages[8].iIndex := 230;
		aTransferPackages[8].iTransferValue := iOptProportionalGainFor2;
	
	//iOptIntegralGainFor2
		aTransferPackages[9].iChannel := iParameterSet;
		aTransferPackages[9].iAddressedTarget := 10;
		aTransferPackages[9].iIndex := 231;
		aTransferPackages[9].iTransferValue := iOptIntegralGainFor2;
	
	//iOptRedFeedforwContrRate2
		aTransferPackages[10].iChannel := iParameterSet;
		aTransferPackages[10].iAddressedTarget := 10;
		aTransferPackages[10].iIndex := 232;
		aTransferPackages[10].iTransferValue := iOptRedFeedforwContrRate2;
	
	//iOptBoostSetpointReach2
		aTransferPackages[11].iChannel := iParameterSet;
		aTransferPackages[11].iAddressedTarget := 10;
		aTransferPackages[11].iIndex := 233;
		aTransferPackages[11].iTransferValue := iOptBoostSetpointReach2;
	
	//iOptOffsetTargFRLimitInfo2
		aTransferPackages[12].iChannel := iParameterSet;
		aTransferPackages[12].iAddressedTarget := 10;
		aTransferPackages[12].iIndex := 234;
		aTransferPackages[12].iTransferValue := iOptOffsetTargFRLimitInfo2;
	
	//iOptOffsetMinConsSetp2
		aTransferPackages[13].iChannel := iParameterSet;
		aTransferPackages[13].iAddressedTarget := 10;
		aTransferPackages[13].iIndex := 235;
		aTransferPackages[13].iTransferValue := iOptOffsetMinConsSetp2;
	
	//iOptProportionalGainFor4
		aTransferPackages[14].iChannel := iParameterSet;
		aTransferPackages[14].iAddressedTarget := 10;
		aTransferPackages[14].iIndex := 240;
		aTransferPackages[14].iTransferValue := iOptProportionalGainFor4;
	
	//iOptIntegralGainFor4
		aTransferPackages[15].iChannel := iParameterSet;
		aTransferPackages[15].iAddressedTarget := 10;
		aTransferPackages[15].iIndex := 241;
		aTransferPackages[15].iTransferValue := iOptIntegralGainFor4;
	
	//iOptRedFeedforwContrRate4
		aTransferPackages[16].iChannel := iParameterSet;
		aTransferPackages[16].iAddressedTarget := 10;
		aTransferPackages[16].iIndex := 242;
		aTransferPackages[16].iTransferValue := iOptRedFeedforwContrRate4;
	
	//iOptBoostSetpointReach4
		aTransferPackages[17].iChannel := iParameterSet;
		aTransferPackages[17].iAddressedTarget := 10;
		aTransferPackages[17].iIndex := 243;
		aTransferPackages[17].iTransferValue := iOptBoostSetpointReach4;
	
	//iOptOffsetTargFRLimitInfo4
		aTransferPackages[18].iChannel := iParameterSet;
		aTransferPackages[18].iAddressedTarget := 10;
		aTransferPackages[18].iIndex := 244;
		aTransferPackages[18].iTransferValue := iOptOffsetTargFRLimitInfo4;
	
	//iOptOffsetMinConsSetp4
		aTransferPackages[19].iChannel := iParameterSet;
		aTransferPackages[19].iAddressedTarget := 10;
		aTransferPackages[19].iIndex := 245;
		aTransferPackages[19].iTransferValue := iOptOffsetMinConsSetp4;
	
	// define end of parameter list to be downloaded by setting all variables to 0 (end criterion for FB_Download_Multiple_Parameters)
		aTransferPackages[20].iChannel := 0;
		aTransferPackages[20].iAddressedTarget := 0;
		aTransferPackages[20].iIndex := 0;
		aTransferPackages[20].iTransferValue := 0;


// pre-check of the value for the parameter set
	IF xExecute = TRUE AND (iParameterSet < 1 OR iParameterSet > 5) THEN		// invalid input for the parameter set
		xDownloadDone := FALSE; 
		xDownloadError := TRUE; 
		iResponse := eTransferResponse.invalid_ParameterSet; 
		iCurrentValue := 0; 
		// send command 'stop'
		fbWriteValueToWord(iValue := 61, iStartBit := 0, iEndBit := 5, wDataWord := awBusDataToVTEM[0]); 			// ValveMode = 61
		fbWriteValueToWord(iValue := 0, iStartBit := 6, iEndBit := 15, wDataWord := awBusDataToVTEM[0]); 			// (empty)
		awBusDataToVTEM[1] := 0; 
		awBusDataToVTEM[2] := 0; 
		
	ELSE	
		// call the function block for multiple parameter download
			fbdownloadMultipleParameters(	xExecute := xExecute,
											awBusDataFromVTEM := awBusDataFromVTEM,
											aTransferPackages := aTransferPackages, 
											awBusDataToVTEM := awBusDataToVTEM,
											xDownloadDone => xDownloadDone,
											xDownloadError => xDownloadError,
											iResponse => iResponse,
											iCurrentValue => iCurrentValue);
	END_IF
	
	
// The current value output is needed if there is any invalid value in order to address it correctly.
// As the user doesn't work with indices in this function block, the current value is transformed to a string holding the name of the parameter.
	CASE iCurrentValue OF
		0: sCurrentValue := 'iOperatingMedium';
		1: sCurrentValue := 'iInPortFlowRate2_optional';
		2: sCurrentValue := 'iInPortFlowRate4_optional';
		3: sCurrentValue := 'iInPortRetracted_optional';
		4: sCurrentValue := 'iInPortAdvanced_optional';
		5: sCurrentValue := 'iCharacteristicAt2';
		6: sCurrentValue := 'iCharacteristicAt4';
		7: sCurrentValue := 'iOperatingMode';
		8: sCurrentValue := 'iOptProportionalGainFor2';
		9: sCurrentValue := 'iOptIntegralGainFor2';
		10: sCurrentValue := 'iOptRedFeedforwContrRate2';
		11: sCurrentValue := 'iOptBoostSetpointReach2';
		12: sCurrentValue := 'iOptOffsetTargFRLimitInfo2';
		13: sCurrentValue := 'iOptOffsetMinConsSetp2';
		14: sCurrentValue := 'iOptProportionalGainFor4';
		15: sCurrentValue := 'iOptIntegralGainFor4';
		16: sCurrentValue := 'iOptRedFeedforwContrRate4';
		17: sCurrentValue := 'iOptBoostSetpointReach4';
		18: sCurrentValue := 'iOptOffsetTargFRLimitInfo4';
		19: sCurrentValue := 'iOptOffsetMinConsSetp4';
		20: sCurrentValue := 'AllParametersWritten';
	END_CASE

END_FUNCTION_BLOCK

// StateInterpreter/FB_StateInterpreter_MA_10
/// The variable "byActualAppState" is an output of the FB_ValveControl that is used differently in each Motion App.
/// This function block interprets the "AppState" output of the FB_ValveControl if Motion App 10 ("Flow control") is running.
/// The Motion App specific values are derived from the "byActualAppState".

FUNCTION_BLOCK FB_StateInterpreter_MA_10
VAR_INPUT
	byActualAppState 			: BYTE; 	(* output of the FB_ValveControl *)
END_VAR
VAR_OUTPUT
	x2or4outOfSpec				: BOOL;		// indicates that port (2) and/or (4) is operated outside the specification
	xFlow2FromMeasurement		: BOOL;		// indicates that actual value for flow on (2) comes from measurement (higher accuracy)
	xFlow4FromMeasurement		: BOOL;		// indicates that actual value for flow on (4) comes from measurement (higher accuracy)
	xRatioSetToMaxOverLimit2	: BOOL;		// Indicates that the ratio of the set flow to the maximum adjustable flow at port (2) is greater than the specified limit (95% of the maximum adjustable flow + value of parameter "iOptOffsetTargFRLimitInfo2")
	xRatioSetToMaxOverLimit4	: BOOL;		// Indicates that the ratio of the set flow to the maximum adjustable flow at port (4) is greater than the specified limit (95% of the maximum adjustable flow + value of parameter "iOptOffsetTargFRLimitInfo4")
	xRetractedEndPos_optional	: BOOL;  	(* only if digital sensors are installed (optional): indicates whether the retracted end position was reached (after outlet port 2 is pressurised) *)
	xAdvancedEndPos_optional	: BOOL;  	(* only if digital sensors are installed (optional): indicates whether the advanced end position was reached (after outlet port 4 is pressurised) *)
	xWarning					: BOOL; 	(* indicates whether there is a warning returned by the Motion App *)
END_VAR
VAR
	fbReadBitsFromByte			: FB_Read_Bits_From_Byte;
	by2or4outOfSpec				: BYTE;
	byFlow2FromMeasurement		: BYTE;	
	byFlow4FromMeasurement		: BYTE;	
	byRatioSetToMaxOverLimit2	: BYTE;	
	byRatioSetToMaxOverLimit4	: BYTE;
	byRetractedEndPos			: BYTE;
	byAdvancedEndPos			: BYTE;
	byWarning					: BYTE;
END_VAR

(*****************************************************************************************************

Festo SE & Co. KG, Esslingen
Copyright (c) 2020. All rights reserved.

Product:            Motion Terminal VTEM
Description:        Function block for interpreting the app state of Motion App 10 

Object version:     1.00
Last change:        2020-11
======================================================================================================
                                       H I S T O R Y
======================================================================================================
Version:            1.00
Date:               2020-11
Change/Activity:    - created (#3805730)
Release:            3.5.7.236
Author:             JEBU
======================================================================================================

*****************************************************************************************************)

// read the Motion App specific values from the ActualAppState byte
fbReadBitsFromByte(byData := byActualAppState, iStartBit := 1, iEndBit := 1, byValue => by2or4outOfSpec);
x2or4outOfSpec :=  BYTE_TO_BIT(by2or4outOfSpec);

fbReadBitsFromByte(byData := byActualAppState, iStartBit := 3, iEndBit := 3, byValue => byFlow2FromMeasurement);
xFlow2FromMeasurement :=  BYTE_TO_BIT(byFlow2FromMeasurement);

fbReadBitsFromByte(byData := byActualAppState, iStartBit := 4, iEndBit := 4, byValue => byFlow4FromMeasurement);
xFlow4FromMeasurement :=  BYTE_TO_BIT(byFlow4FromMeasurement);

fbReadBitsFromByte(byData := byActualAppState, iStartBit := 5, iEndBit := 5, byValue => byRatioSetToMaxOverLimit2);
xRatioSetToMaxOverLimit2 :=  BYTE_TO_BIT(byRatioSetToMaxOverLimit2);

fbReadBitsFromByte(byData := byActualAppState, iStartBit := 6, iEndBit := 6, byValue => byRatioSetToMaxOverLimit4);
xRatioSetToMaxOverLimit4 :=  BYTE_TO_BIT(byRatioSetToMaxOverLimit4);

fbReadBitsFromByte(byData := byActualAppState, iStartBit := 0, iEndBit := 0, byValue => byRetractedEndPos);
xRetractedEndPos_optional :=  BYTE_TO_BIT(byRetractedEndPos);

fbReadBitsFromByte(byData := byActualAppState, iStartBit := 2, iEndBit := 2, byValue => byAdvancedEndPos); 
xAdvancedEndPos_optional :=  BYTE_TO_BIT(byAdvancedEndPos);

fbReadBitsFromByte(byData := byActualAppState, iStartBit := 7, iEndBit := 7, byValue => byWarning);
xWarning := BYTE_TO_BIT(byWarning);

END_FUNCTION_BLOCK

// Operation/FB_AppOptionGenerator_MA_02
/// The App Option byte of Motion App 02 ("Proportional directional control valve") contains several pieces of information.
/// The individual pieces of information can be passed to this function block and it generates the corresponding value for the App Option byte from this.
/// The generated App Option byte can be passed to the FB_ValveControl block.

FUNCTION_BLOCK FB_AppOptionGenerator_MA_02
VAR_INPUT
	usiValveType			: USINT;		// Defines used valve type (14 = 4/3 G (normally closed), 15 = 2 × 3/3nG (normally closed))
	xSetMeaningOfActVal1	: BOOL;			// Setting the meaning of actual value 1 (0 = valve position, 1 = relative pressure)
	xSetMeaningOfActVal2	: BOOL;			// Setting the meaning of actual value 2 (0 = valve position, 1 = relative pressure)
END_VAR
VAR_OUTPUT
	byAppOption				: BYTE;			// AppOption byte to connect with the byAppOption input of FB_ValveControl
END_VAR
VAR
END_VAR

(*****************************************************************************************************

Festo SE & Co. KG, Esslingen
Copyright (c) 2021. All rights reserved.

Product:            Motion Terminal VTEM
Description:        Function block for generating the app option byte for Motion App 2

Object version:     1.00
Last change:        2021-01
======================================================================================================
                                       H I S T O R Y
======================================================================================================
Version:            1.00
Date:               2021-01
Change/Activity:    - created (#3919898)
Release:            3.5.7.236
Author:             JEBU
======================================================================================================

*****************************************************************************************************)
IF usiValveType >= 14 AND usiValveType <= 15 THEN
	byAppOption := USINT_TO_BYTE(usiValveType);
	byAppOption.5 := xSetMeaningOfActVal1;
	byAppOption.6 := xSetMeaningOfActVal2;	
ELSE
	byAppOption := 0;
END_IF

END_FUNCTION_BLOCK

// Transfermode/specific_MA_config/FB_Read_config_MA_01
/// This function block can be used to upload the configuration of Motion App 1 ("Directional control valve functions").
/// The specific parameters of this Motion App are the outputs of this FB
/// The function block uses the transfer mode to read this configuration from the Motion Terminal
/// and indicates the state of the upload process at the output iResponse.

FUNCTION_BLOCK FB_Read_config_MA_01
VAR_INPUT
	awBusDataFromVTEM 				: ARRAY [0..2] OF WORD;		// array of 3 words of process data received from the Motion Terminal
END_VAR
	
VAR_IN_OUT
	awBusDataToVTEM 				: ARRAY [0..2] OF WORD; 	// array of 3 words of process data sent to the Motion Terminal
END_VAR

VAR_INPUT
	xExecute 						: BOOL; 					// rising edge starts the reading process, falling edge resets the function block after reading is done
	xAbort							: BOOL;						// rising edge aborts the reading process
	iParameterSet					: INT := 1; 				// the parameter set to be read from, 1 by default
END_VAR                     		

VAR_OUTPUT                  		
	// application parameters
		iOperatingMode				: INT := 0;	 				// Switching the operating mode (0 = open loop controlled, 1 = close-loop controlled) 
	// system parameters
		iInPortRetracted_optional	: INT;						// Sensor port for detection of end position at pressurisation of outlet port 2 (retracted), value is number of the slot (beginning from 0 and including valve slots) * 10 + number of the port
		iInPortAdvanced_optional	: INT;						// Sensor port for detection of end position at pressurisation of outlet port 4 (advanced), value is number of the slot (beginning from 0 and including valve slots) * 10 + number of the port
	// function block response
		iResponse 					: eTransferResponse; 		// returns the status of the upload process
		xBusy						: BOOL;						// TRUE as long as the upload process is running
		xDone 						: BOOL; 					// indicates whether the upload was successfull
		xError 						: BOOL; 					// indicates whether an error occurred during the transfer
		xAborted					: BOOL;						// TRUE if the function block was canceled by xAbort
END_VAR

VAR
	iState							: INT := 10;
	xStateChange					: BOOL;
	iCommandNumber					: INT;
	xFirstCycle						: BOOL := TRUE;				// indicator for the first cycle of the function block
	iParameterSetFC					: INT;						// value on input iParameterSet during first cycle
	
	aTransferPackages				: ARRAY [0..100] OF stTransferPackage;
	fbreadbitsfromword				: FB_Read_Bits_From_Word;
	fbuploadMultipleParameters 		: FB_Upload_Multiple_Parameters;
	fbWriteValueToWord 				: FB_Write_Value_To_Word;
	
	iCounterResetArray				: INT;
	
	iCurrentValveMode				: INT;						//
END_VAR

(*****************************************************************************************************

Festo SE & Co. KG, Esslingen
Copyright (c) 2021. All rights reserved.

Product:            Motion Terminal VTEM
Description:        Function Block to upload the parameters for Motion App 1 from the Motion Terminal

Object version:     2.00
Last change:        2021-07
======================================================================================================
                                       H I S T O R Y
======================================================================================================
Version:            2.00
Date:               2021-07
Change/Activity:    - created (#3872357)
Release:            3.5.7.237 (CODESYS 3.5.7.2, Lib version 3.7)
Author:             JEBU
======================================================================================================

*****************************************************************************************************)

// pre-check of the value for the parameter set
	IF xExecute = TRUE AND (iParameterSet < 1 OR iParameterSet > 5) THEN		// invalid input for the parameter set
		xDone := FALSE; 
		xError := TRUE; 
		iResponse := eTransferResponse.invalid_ParameterSet;
		xStateChange := TRUE;
		iState := 70;	// ERROR
	END_IF
//-----------------------------------------------------------------------------------------------------------

// check if iParameterSet was changed
	IF xExecute = TRUE AND xFirstCycle = TRUE THEN
		xFirstCycle := FALSE;
		iParameterSetFC := iParameterSet;
	END_IF
	
	IF xExecute = TRUE AND iParameterSet <> iParameterSetFC THEN
		xStateChange := TRUE;
		iState := 70;
		iResponse := eTransferResponse.FB_needs_rising_edge_xExecute;
	END_IF
//-----------------------------------------------------------------------------------------------------------

// WRITE PARAMETER INDICES INTO ARRAY
	//iOperatingMode
		aTransferPackages[0].iChannel := iParameterSet;
		aTransferPackages[0].iAddressedTarget := 1;
		aTransferPackages[0].iIndex := 223;
	
	//iInPortRetract_optional
		aTransferPackages[1].iChannel := iParameterSet;
		aTransferPackages[1].iAddressedTarget := 1;
		aTransferPackages[1].iIndex := 70;
	
	//iInPortRetract_optional
		aTransferPackages[2].iChannel := iParameterSet;
		aTransferPackages[2].iAddressedTarget := 1;
		aTransferPackages[2].iIndex := 71;
	
	// define end of parameter list to be uploaded by setting all variables to 0 (end criterion for FB_Upload_Multiple_Parameters)
		aTransferPackages[3].iChannel := 0;
		aTransferPackages[3].iAddressedTarget := 0;
		aTransferPackages[3].iIndex := 0;
//-----------------------------------------------------------------------------------------------------------

// Read the current status of the the motion terminal
	fbreadbitsfromword(wData:= awBusDataFromVTEM[0], iStartBit:=0, iEndBit:= 5, iValue=> iCurrentValveMode, xError=> );				// read current valve mode
//-----------------------------------------------------------------------------------------------------------

// Transition: Aborting condition when xAbort is TRUE in all States except "IDLE" , "ABORTING" and "RESETTING"
	IF xAbort = TRUE AND NOT(iState = 10 AND xExecute = FALSE) AND iState <> 80 AND iState <> 100 THEN
		xStateChange := TRUE;	// Leaving current state
		iState := 80;	// Choosing next state, here: ABORTING
	END_IF
//-----------------------------------------------------------------------------------------------------------

// local state machine
	CASE iState OF
		10:	// IDLE
			// code that is executed only in the first cycle of this state
				IF xStateChange = TRUE THEN
					xStateChange := FALSE;
					iResponse := eTransferResponse.ready_for_new_transfer;
					xDone := FALSE;
					xError := FALSE;
					xBusy := FALSE;
					xAborted := FALSE;
				END_IF
			//-----------------------------------------------------------------------------------------------------------
			
			// code that is repeated every cycle in this state
				iCommandNumber := 0;
			//-----------------------------------------------------------------------------------------------------------
			
			// Transition
			IF xExecute = TRUE THEN
				xStateChange := TRUE;
				iState := 20;
			END_IF
			//-----------------------------------------------------------------------------------------------------------
		
		20:	// RESETTING VALVE MODE TO 61
			// code that is executed only in the first cycle of this state
				IF xStateChange = TRUE THEN
					xStateChange := FALSE;
					iResponse := eTransferResponse.preparing_transfer;
					xDone := FALSE;
					xError := FALSE;
					xBusy := TRUE;
					xAborted := FALSE;
				END_IF
			//-----------------------------------------------------------------------------------------------------------
			
			// code that is repeated every cycle in this state	
				IF iCurrentValveMode = 63 THEN
					iCommandNumber := 5;	// exit transfer mode
				ELSIF iCurrentValveMode <> 61 AND iCurrentValveMode <> 63 THEN
					iCommandNumber := 6;	// stop running motion apps
				END_IF 
			//-----------------------------------------------------------------------------------------------------------
			
			// Transition
				IF iCurrentValveMode = 61 THEN
					xStateChange := TRUE;	// Leave this state
					iState := 30;
					iCommandNumber := 30;			
				END_IF
			//-----------------------------------------------------------------------------------------------------------
		
		30:	// READING PARAMETER VALUES
			// code that is executed only in the first cycle of this state
				IF xStateChange = TRUE THEN
					xStateChange := FALSE;
					iResponse := eTransferResponse.transferring;
					xDone := FALSE;
					xError := FALSE;
					xBusy := TRUE;
					xAborted := FALSE;
				END_IF
			//-----------------------------------------------------------------------------------------------------------
			
			// code that is repeated every cycle in this state
				iCommandNumber := 30;		// read parameter values
			//-----------------------------------------------------------------------------------------------------------
			
			// Transition
				IF fbuploadMultipleParameters.xExecute = TRUE AND fbuploadMultipleParameters.xUploadDone = TRUE AND fbuploadMultipleParameters.xUploadError = FALSE THEN	// Upload Done
					xStateChange := TRUE;
					iState := 40;	// Write parameter values to outputs
				ELSIF fbuploadMultipleParameters.xExecute = TRUE AND fbuploadMultipleParameters.xUploadDone = FALSE AND fbuploadMultipleParameters.xUploadError = TRUE THEN	// Error during update
					xStateChange := TRUE;
					iState := 70;	// ERROR
					iResponse := fbuploadMultipleParameters.iResponse;
				END_IF
			//-----------------------------------------------------------------------------------------------------------
		
		40:	// WRITE PARAMETER VALUES TO OUTPUTS
			// code that is executed only in the first cycle of this state
				IF xStateChange = TRUE THEN
					xStateChange := FALSE;
					iResponse := eTransferResponse.transferring;
					xDone := FALSE;
					xError := FALSE;
					xBusy := TRUE;
					xAborted := FALSE;
				END_IF
			//-----------------------------------------------------------------------------------------------------------
			
			// code that is repeated every cycle in this state
				iOperatingMode				:= aTransferPackages[0].iTransferValue;
				iInPortRetracted_optional	:= aTransferPackages[1].iTransferValue;
				iInPortAdvanced_optional	:= aTransferPackages[2].iTransferValue;
			//-----------------------------------------------------------------------------------------------------------
			
			// Transition
				xStateChange := TRUE;
				iState := 50;
				iCommandNumber := 40;
			//-----------------------------------------------------------------------------------------------------------
		
		50:	// DONE
			// code that is executed only in the first cycle of this state
				IF xStateChange = TRUE THEN
					xStateChange := FALSE;
					iResponse := eTransferResponse.transfer_successful;
					xDone := TRUE;
					xError := FALSE;
					xBusy := FALSE;
					xAborted := FALSE;
				END_IF
			//-----------------------------------------------------------------------------------------------------------
			
			// code that is repeated every cycle in this state	
				IF fbuploadMultipleParameters.xExecute = FALSE  AND fbuploadMultipleParameters.xUploadDone = FALSE AND fbuploadMultipleParameters.xUploadError = FALSE AND iCurrentValveMode = 63 THEN		//FB_UploadMultipleParameters was reset
					iCommandNumber := 5;	// exit transfer mode
				END_IF
			//-----------------------------------------------------------------------------------------------------------
			
			// Transition
				IF fbuploadMultipleParameters.xExecute = FALSE  AND fbuploadMultipleParameters.xUploadDone = FALSE AND fbuploadMultipleParameters.xUploadError = FALSE AND xExecute = FALSE THEN
					xStateChange := TRUE;
					iState := 100;
				END_IF
			//-----------------------------------------------------------------------------------------------------------
			
		70:	// ERROR
			// code that is executed only in the first cycle of this state
				IF xStateChange = TRUE THEN
					xStateChange := FALSE;
					//iResponse := ;	// set within the transition of the last state
					xDone := FALSE;
					xError := TRUE;
					xBusy := FALSE;
					xAborted := FALSE;
				END_IF
			//-----------------------------------------------------------------------------------------------------------
			
			// code that is repeated every cycle in this state	
			//-----------------------------------------------------------------------------------------------------------
			
			// Transition
				IF xExecute = FALSE AND xAbort = FALSE THEN
					xStateChange := TRUE;
					iState := 100;
				END_IF
			//-----------------------------------------------------------------------------------------------------------
			
		80:	// ABORTING
			// code that is executed only in the first cycle of this state
				IF xStateChange = TRUE THEN
					xStateChange := FALSE;
					iResponse := eTransferResponse.aborting;
					xBusy := FALSE;
					xDone := FALSE;
					xError := FALSE;
					xAborted := TRUE;
				END_IF
			//-----------------------------------------------------------------------------------------------------------
			
			// code that is repeated every cycle in this state
				IF iCurrentValveMode = 63 THEN
					iCommandNumber := 5;	// exit transfer mode
				ELSIF iCurrentValveMode <> 61 AND iCurrentValveMode <> 63 THEN
					iCommandNumber := 6;	// stop running motion apps
				ELSE
					iCommandNumber := 0; 
				END_IF
			//-----------------------------------------------------------------------------------------------------------
			
			// Transition
				IF xAbort = FALSE AND xExecute = FALSE AND iCurrentValveMode = 61 THEN
					xStateChange := TRUE;
					iState := 100;
				END_IF
			//-----------------------------------------------------------------------------------------------------------

		100:	// RESETTING FUNCTION BLOCK AND VALVE
			// code that is executed only in the first cycle of this state
				IF xStateChange = TRUE THEN
					xStateChange := FALSE;
					iResponse := eTransferResponse.resetting;
					xDone := FALSE;
					xError := FALSE;
					xBusy := FALSE;
					xAborted := FALSE;
				END_IF
			//-----------------------------------------------------------------------------------------------------------
			
			// code that is repeated every cycle in this state	
				IF iCurrentValveMode = 63 THEN
					iCommandNumber := 5;	// exit transfer mode
				ELSIF iCurrentValveMode <> 61 AND iCurrentValveMode <> 63 THEN
					iCommandNumber := 6;	// stop running motion apps
				END_IF
				
				// reset funktion block fbreadmultipleparameters
				// not done via command number because this is used to reset valve
					fbuploadMultipleParameters(
						awBusDataFromVTEM:= awBusDataFromVTEM, 
						awBusDataToVTEM:= awBusDataToVTEM, 
						xExecute:= FALSE, 
						iResponse=> , 
						iCurrentValue=> , 
						xUploadDone=> , 
						xUploadError=> , 
						aTransferPackages:= aTransferPackages);
				
				// reset parameter outputs
					iParameterSet := 1;
					iOperatingMode := 0;
					iInPortRetracted_optional := 0;
					iInPortAdvanced_optional := 0;
				
				// reset parameter array
					FOR iCounterResetArray := 0 TO 100 BY 1 DO
						aTransferPackages[iCounterResetArray].iChannel := 0;
						aTransferPackages[iCounterResetArray].iAddressedTarget := 0;
						aTransferPackages[iCounterResetArray].iIndex := 0;
						aTransferPackages[iCounterResetArray].iTransferValue := 0;
					END_FOR
					
					iCounterResetArray := 0;
					xFirstCycle := TRUE;
			//-----------------------------------------------------------------------------------------------------------
			
			// Transition
				IF iCurrentValveMode = 61 THEN
					iCommandNumber := 6; // Last command to send before the FB is in IDLE
					xStateChange := TRUE;
					iState := 10;
				END_IF
			//-----------------------------------------------------------------------------------------------------------
			
	END_CASE
//-----------------------------------------------------------------------------------------------------------

// Command section
	CASE iCommandNumber OF
		0:	// IDLE
			;
		
		5:	// EXIT TRANSFER MODE
			fbwritevaluetoword(iValue:=63, iStartBit:=0, iEndBit:=5, wDataWord:=awBusDataToVTEM[0], xError=> );							// Valve Mode = 63
			fbwritevaluetoword(iValue:=0, iStartBit:=6, iEndBit:=7, wDataWord:=awBusDataToVTEM[0], xError=> );							// 0 (unused)
			fbwritevaluetoword(iValue:=0, iStartBit:=8, iEndBit:=12, wDataWord:=awBusDataToVTEM[0], xError=> );							// Channel = 0 (ignored)
			fbwritevaluetoword(iValue:=3, iStartBit:=13, iEndBit:=15, wDataWord:=awBusDataToVTEM[0], xError=> );						// Transfer Control = 3 (Exit transfer mode)
			fbwritevaluetoword(iValue:=0, iStartBit:=0, iEndBit:=7, wDataWord:=awBusDataToVTEM[1], xError=> );							// Addressed Target = 0 (ignored)
			fbwritevaluetoword(iValue:=0, iStartBit:=8, iEndBit:=15, wDataWord:=awBusDataToVTEM[1], xError=> );							// Index = 0 (ignored)
			fbwritevaluetoword(iValue:=0, iStartBit:=0, iEndBit:=15, wDataWord:=awBusDataToVTEM[2], xError=> );							// Value = 0 (ignored)
			
		6:	// STOP RUNNING MOTION APP
			fbwritevaluetoword(iValue:=61, iStartBit:=0, iEndBit:=5, wDataWord:=awBusDataToVTEM[0], xError=> );							// Valve Mode = 61 (stop)
			fbwritevaluetoword(iValue:=0, iStartBit:=6, iEndBit:=7, wDataWord:=awBusDataToVTEM[0], xError=> );							// App Control = 0 (unused)
			fbwritevaluetoword(iValue:=0, iStartBit:=8, iEndBit:=15, wDataWord:=awBusDataToVTEM[0], xError=> );							// App Option = 0 (unused)
			fbwritevaluetoword(iValue:=0, iStartBit:=0, iEndBit:=15, wDataWord:=awBusDataToVTEM[1], xError=> );							// Setpoint Value 1 = 0 (unused)
			fbwritevaluetoword(iValue:=0, iStartBit:=0, iEndBit:=15, wDataWord:=awBusDataToVTEM[2], xError=> );							// Setpoint Value 2 = 0 (unused)
		
		30:	// RUN FB_UPLOADMULTIPLEPARAMETERS
			fbuploadMultipleParameters(
				awBusDataFromVTEM:= awBusDataFromVTEM, 
				awBusDataToVTEM:= awBusDataToVTEM, 
				xExecute:= TRUE, 
				iResponse=> , 
				iCurrentValue=> , 
				xUploadDone=> , 
				xUploadError=> , 
				aTransferPackages:= aTransferPackages);

		40:	// RESET FB_UPLOADMULTIPLEPARAMETERS
			fbuploadMultipleParameters(
				awBusDataFromVTEM:= awBusDataFromVTEM, 
				awBusDataToVTEM:= awBusDataToVTEM, 
				xExecute:= FALSE, 
				iResponse=> , 
				iCurrentValue=> , 
				xUploadDone=> , 
				xUploadError=> , 
				aTransferPackages:= aTransferPackages);
	END_CASE
//-----------------------------------------------------------------------------------------------------------

END_FUNCTION_BLOCK

// Transfermode/specific_MA_config/FB_Read_config_MA_02
/// This function block can be used to upload the configuration of Motion App 2 ("Proportional directional control valve").
/// The specific parameters of this Motion App are the outputs of this FB
/// The function block uses the transfer mode to read this configuration from the Motion Terminal
/// and indicates the state of the upload process at the output iResponse.

FUNCTION_BLOCK FB_Read_config_MA_02
VAR_INPUT
	awBusDataFromVTEM 				: ARRAY [0..2] OF WORD;		// array of 3 words of process data received from the Motion Terminal
END_VAR
	
VAR_IN_OUT
	awBusDataToVTEM 				: ARRAY [0..2] OF WORD; 	// array of 3 words of process data sent to the Motion Terminal
END_VAR

VAR_INPUT
	xExecute 						: BOOL; 					// rising edge starts the reading process, falling edge resets the function block after reading is done
	xAbort							: BOOL;						// rising edge aborts the reading process
	iParameterSet					: INT := 1; 				// the parameter set to be read from, 1 by default
END_VAR                     		

VAR_OUTPUT                  		
	// system parameters
		iInPortRetracted_optional	: INT;						// Sensor port for detection of end position at pressurisation of outlet port 2 (retracted), value is number of the slot (beginning from 0 and including valve slots) * 10 + number of the port
		iInPortAdvanced_optional	: INT;						// Sensor port for detection of end position at pressurisation of outlet port 4 (advanced), value is number of the slot (beginning from 0 and including valve slots) * 10 + number of the port
		
	// application parameters
		iCharacteristicAt2 			: INT; 						// characteristic of the control algorithm for outlet port 2 (0 = precise, 1 = universal, 2 = fast)
		iCharacteristicAt4 			: INT; 						// characteristic of the control algorithm for outlet port 4 (0 = precise, 1 = universal, 2 = fast)
		iOperatingMode				: INT;	 					// Switching the operating mode (0 = seal seat behaviour, 1 = servo mode)
		
	// function block response
		iResponse 					: eTransferResponse; 		// returns the status of the upload process
		xBusy						: BOOL;						// TRUE as long as the upload process is running
		xDone 						: BOOL; 					// indicates whether the upload was successfull
		xError 						: BOOL; 					// indicates whether an error occurred during the transfer
		xAborted					: BOOL;						// TRUE if the function block was canceled by xAbort	
END_VAR

VAR
	iState							: INT := 10;
	xStateChange					: BOOL;
	iCommandNumber					: INT;
	xFirstCycle						: BOOL := TRUE;				// indicator for the first cycle of the function block
	iParameterSetFC					: INT;						// value on input iParameterSet during first cycle
	
	aTransferPackages				: ARRAY [0..100] OF stTransferPackage;
	fbreadbitsfromword				: FB_Read_Bits_From_Word;
	fbuploadMultipleParameters 		: FB_Upload_Multiple_Parameters;
	fbWriteValueToWord 				: FB_Write_Value_To_Word;

	iCounterResetArray				: INT;

	iCurrentValveMode				: INT;						//
END_VAR

(*****************************************************************************************************

Festo SE & Co. KG, Esslingen
Copyright (c) 2021. All rights reserved.

Product:            Motion Terminal VTEM
Description:        Function Block to upload the parameters for Motion App 2 from the Motion Terminal

Object version:     2.00
Last change:        2021-07
======================================================================================================
                                       H I S T O R Y
======================================================================================================
Version:            2.00
Date:               2021-07
Change/Activity:    - created (#3872357)
Release:            3.5.7.237 (CODESYS 3.5.7.2, Lib version 3.7)
Author:             JEBU
======================================================================================================

*****************************************************************************************************)

// pre-check of the value for the parameter set
	IF xExecute = TRUE AND (iParameterSet < 1 OR iParameterSet > 5) THEN		// invalid input for the parameter set
		xDone := FALSE; 
		xError := TRUE; 
		iResponse := eTransferResponse.invalid_ParameterSet;
		xStateChange := TRUE;
		iState := 70;	// ERROR
	END_IF
//-----------------------------------------------------------------------------------------------------------

// check if iParameterSet was changed
	IF xExecute = TRUE AND xFirstCycle = TRUE THEN
		xFirstCycle := FALSE;
		iParameterSetFC := iParameterSet;
	END_IF
	
	IF xExecute = TRUE AND iParameterSet <> iParameterSetFC THEN
		xStateChange := TRUE;
		iState := 70;
		iResponse := eTransferResponse.FB_needs_rising_edge_xExecute;
	END_IF
//-----------------------------------------------------------------------------------------------------------

// WRITE PARAMETER INDICES INTO ARRAY
	//iCharacteristicAt2
		aTransferPackages[0].iChannel := iParameterSet;
		aTransferPackages[0].iAddressedTarget := 2;
		aTransferPackages[0].iIndex := 220;
	
	//iCharacteristicAt4
		aTransferPackages[1].iChannel := iParameterSet;
		aTransferPackages[1].iAddressedTarget := 2;
		aTransferPackages[1].iIndex := 221;
	
	//iInPortRetract_optional
		aTransferPackages[2].iChannel := iParameterSet;
		aTransferPackages[2].iAddressedTarget := 2;
		aTransferPackages[2].iIndex := 70;
	
	//iInPortAdvanced_optional
		aTransferPackages[3].iChannel := iParameterSet;
		aTransferPackages[3].iAddressedTarget := 2;
		aTransferPackages[3].iIndex := 71;
	
	//iOperatingMode
		aTransferPackages[4].iChannel := iParameterSet;
		aTransferPackages[4].iAddressedTarget := 2;
		aTransferPackages[4].iIndex := 223;
	
	// define end of parameter list to be uploaded by setting all variables to 0 (end criterion for FB_Upload_Multiple_Parameters)
		aTransferPackages[5].iChannel := 0;
		aTransferPackages[5].iAddressedTarget := 0;
		aTransferPackages[5].iIndex := 0;
//-----------------------------------------------------------------------------------------------------------

// Read the current status of the the motion terminal
	fbreadbitsfromword(wData:= awBusDataFromVTEM[0], iStartBit:=0, iEndBit:= 5, iValue=> iCurrentValveMode, xError=> );				// read current valve mode
//-----------------------------------------------------------------------------------------------------------

// Transition: Aborting condition when xAbort is TRUE in all States except "IDLE" , "ABORTING" and "RESETTING"
	IF xAbort = TRUE AND NOT(iState = 10 AND xExecute = FALSE) AND iState <> 80 AND iState <> 100 THEN
		xStateChange := TRUE;	// Leaving current state
		iState := 80;	// Choosing next state, here: ABORTING
	END_IF
//-----------------------------------------------------------------------------------------------------------

// local state machine
	CASE iState OF
		10:	// IDLE
			// code that is executed only in the first cycle of this state
				IF xStateChange = TRUE THEN
					xStateChange := FALSE;
					iResponse := eTransferResponse.ready_for_new_transfer;
					xDone := FALSE;
					xError := FALSE;
					xBusy := FALSE;
					xAborted := FALSE;
				END_IF
			//-----------------------------------------------------------------------------------------------------------
			
			// code that is repeated every cycle in this state
				iCommandNumber := 0;
			//-----------------------------------------------------------------------------------------------------------
			
			// Transition
			IF xExecute = TRUE THEN
				xStateChange := TRUE;
				iState := 20;
			END_IF
			//-----------------------------------------------------------------------------------------------------------
		
		20:	// RESETTING VALVE MODE TO 61
			// code that is executed only in the first cycle of this state
				IF xStateChange = TRUE THEN
					xStateChange := FALSE;
					iResponse := eTransferResponse.preparing_transfer;
					xDone := FALSE;
					xError := FALSE;
					xBusy := TRUE;
					xAborted := FALSE;
				END_IF
			//-----------------------------------------------------------------------------------------------------------
			
			// code that is repeated every cycle in this state	
				IF iCurrentValveMode = 63 THEN
					iCommandNumber := 5;	// exit transfer mode
				ELSIF iCurrentValveMode <> 61 AND iCurrentValveMode <> 63 THEN
					iCommandNumber := 6;	// stop running motion apps
				END_IF 
			//-----------------------------------------------------------------------------------------------------------
			
			// Transition
				IF iCurrentValveMode = 61 THEN
					xStateChange := TRUE;	// Leave this state
					iState := 30;
					iCommandNumber := 30;			
				END_IF
			//-----------------------------------------------------------------------------------------------------------
		
		30:	// READING PARAMETER VALUES
			// code that is executed only in the first cycle of this state
				IF xStateChange = TRUE THEN
					xStateChange := FALSE;
					iResponse := eTransferResponse.transferring;
					xDone := FALSE;
					xError := FALSE;
					xBusy := TRUE;
					xAborted := FALSE;
				END_IF
			//-----------------------------------------------------------------------------------------------------------
			
			// code that is repeated every cycle in this state
				iCommandNumber := 30;		// read parameter values
			//-----------------------------------------------------------------------------------------------------------
			
			// Transition
				IF fbuploadMultipleParameters.xExecute = TRUE AND fbuploadMultipleParameters.xUploadDone = TRUE AND fbuploadMultipleParameters.xUploadError = FALSE THEN	// Upload Done
					xStateChange := TRUE;
					iState := 40;	// Write parameter values to outputs
				ELSIF fbuploadMultipleParameters.xExecute = TRUE AND fbuploadMultipleParameters.xUploadDone = FALSE AND fbuploadMultipleParameters.xUploadError = TRUE THEN	// Error during update
					xStateChange := TRUE;
					iState := 70;	// ERROR
					iResponse := fbuploadMultipleParameters.iResponse;
				END_IF
			//-----------------------------------------------------------------------------------------------------------
		
		40:	// WRITE PARAMETER VALUES TO OUTPUTS
			// code that is executed only in the first cycle of this state
				IF xStateChange = TRUE THEN
					xStateChange := FALSE;
					iResponse := eTransferResponse.transferring;
					xDone := FALSE;
					xError := FALSE;
					xBusy := TRUE;
					xAborted := FALSE;
				END_IF
			//-----------------------------------------------------------------------------------------------------------
			
			// code that is repeated every cycle in this state
				iCharacteristicAt2			:= aTransferPackages[0].iTransferValue;
				iCharacteristicAt4			:= aTransferPackages[1].iTransferValue;
				iInPortRetracted_optional	:= aTransferPackages[2].iTransferValue;
				iInPortAdvanced_optional	:= aTransferPackages[3].iTransferValue;
				iOperatingMode				:= aTransferPackages[4].iTransferValue;
			//-----------------------------------------------------------------------------------------------------------
			
			// Transition
				xStateChange := TRUE;
				iState := 50;
				iCommandNumber := 40;
			//-----------------------------------------------------------------------------------------------------------
		
		50:	// DONE
			// code that is executed only in the first cycle of this state
				IF xStateChange = TRUE THEN
					xStateChange := FALSE;
					iResponse := eTransferResponse.transfer_successful;
					xDone := TRUE;
					xError := FALSE;
					xBusy := FALSE;
					xAborted := FALSE;
				END_IF
			//-----------------------------------------------------------------------------------------------------------
			
			// code that is repeated every cycle in this state	
				IF fbuploadMultipleParameters.xExecute = FALSE  AND fbuploadMultipleParameters.xUploadDone = FALSE AND fbuploadMultipleParameters.xUploadError = FALSE AND iCurrentValveMode = 63 THEN		//FB_UploadMultipleParameters was reset
					iCommandNumber := 5;	// exit transfer mode
				END_IF
			//-----------------------------------------------------------------------------------------------------------
			
			// Transition
				IF fbuploadMultipleParameters.xExecute = FALSE  AND fbuploadMultipleParameters.xUploadDone = FALSE AND fbuploadMultipleParameters.xUploadError = FALSE AND xExecute = FALSE THEN
					xStateChange := TRUE;
					iState := 100;
				END_IF
			//-----------------------------------------------------------------------------------------------------------
			
		70:	// ERROR
			// code that is executed only in the first cycle of this state
				IF xStateChange = TRUE THEN
					xStateChange := FALSE;
					//iResponse := eTransferResponse.communication_failed;	// set within the transition of the last state
					xDone := FALSE;
					xError := TRUE;
					xBusy := FALSE;
					xAborted := FALSE;
				END_IF
			//-----------------------------------------------------------------------------------------------------------
			
			// code that is repeated every cycle in this state	
			//-----------------------------------------------------------------------------------------------------------
			
			// Transition
				IF xExecute = FALSE AND xAbort = FALSE THEN
					xStateChange := TRUE;
					iState := 100;
				END_IF
			//-----------------------------------------------------------------------------------------------------------
			
		80:	// ABORTING
			// code that is executed only in the first cycle of this state
				IF xStateChange = TRUE THEN
					xStateChange := FALSE;
					iResponse := eTransferResponse.aborting;
					xBusy := FALSE;
					xDone := FALSE;
					xError := FALSE;
					xAborted := TRUE;
				END_IF
			//-----------------------------------------------------------------------------------------------------------
			
			// code that is repeated every cycle in this state
				IF iCurrentValveMode = 63 THEN
					iCommandNumber := 5;	// exit transfer mode
				ELSIF iCurrentValveMode <> 61 AND iCurrentValveMode <> 63 THEN
					iCommandNumber := 6;	// stop running motion apps
				ELSE
					iCommandNumber := 0; 
				END_IF
			//-----------------------------------------------------------------------------------------------------------
			
			// Transition
				IF xAbort = FALSE AND xExecute = FALSE AND iCurrentValveMode = 61 THEN
					xStateChange := TRUE;
					iState := 100;
				END_IF
			//-----------------------------------------------------------------------------------------------------------

		100:	// RESETTING FUNCTION BLOCK AND VALVE
			// code that is executed only in the first cycle of this state
				IF xStateChange = TRUE THEN
					xStateChange := FALSE;
					iResponse := eTransferResponse.resetting;
					xDone := FALSE;
					xError := FALSE;
					xBusy := FALSE;
					xAborted := FALSE;
				END_IF
			//-----------------------------------------------------------------------------------------------------------
			
			// code that is repeated every cycle in this state	
				IF iCurrentValveMode = 63 THEN
					iCommandNumber := 5;	// exit transfer mode
				ELSIF iCurrentValveMode <> 61 AND iCurrentValveMode <> 63 THEN
					iCommandNumber := 6;	// stop running motion apps
				END_IF
				
				// reset funktion block fbreadmultipleparameters
				// not done via command number because this is used to reset valve
					fbuploadMultipleParameters(
						awBusDataFromVTEM:= awBusDataFromVTEM, 
						awBusDataToVTEM:= awBusDataToVTEM, 
						xExecute:= FALSE, 
						iResponse=> , 
						iCurrentValue=> , 
						xUploadDone=> , 
						xUploadError=> , 
						aTransferPackages:= aTransferPackages);
				
				// reset parameter outputs
					iParameterSet 				:= 1;

					iCharacteristicAt2			:= 0;
					iCharacteristicAt4			:= 0;
					iInPortRetracted_optional	:= 0;
					iInPortAdvanced_optional	:= 0;
					iOperatingMode				:= 0;
				
				// reset parameter array
					FOR iCounterResetArray := 0 TO 100 BY 1 DO
						aTransferPackages[iCounterResetArray].iChannel := 0;
						aTransferPackages[iCounterResetArray].iAddressedTarget := 0;
						aTransferPackages[iCounterResetArray].iIndex := 0;
						aTransferPackages[iCounterResetArray].iTransferValue := 0;
					END_FOR
					
					iCounterResetArray := 0;
					xFirstCycle := TRUE;
			//-----------------------------------------------------------------------------------------------------------
			
			// Transition
				IF iCurrentValveMode = 61 THEN
					iCommandNumber := 6; // Last command to send before the FB is in IDLE
					xStateChange := TRUE;
					iState := 10;
				END_IF
			//-----------------------------------------------------------------------------------------------------------
			
	END_CASE
//-----------------------------------------------------------------------------------------------------------

// Command section
	CASE iCommandNumber OF
		0:	// IDLE
			;
		
		5:	// EXIT TRANSFER MODE
			fbwritevaluetoword(iValue:=63, iStartBit:=0, iEndBit:=5, wDataWord:=awBusDataToVTEM[0], xError=> );							// Valve Mode = 63
			fbwritevaluetoword(iValue:=0, iStartBit:=6, iEndBit:=7, wDataWord:=awBusDataToVTEM[0], xError=> );							// 0 (unused)
			fbwritevaluetoword(iValue:=0, iStartBit:=8, iEndBit:=12, wDataWord:=awBusDataToVTEM[0], xError=> );							// Channel = 0 (ignored)
			fbwritevaluetoword(iValue:=3, iStartBit:=13, iEndBit:=15, wDataWord:=awBusDataToVTEM[0], xError=> );						// Transfer Control = 3 (Exit transfer mode)
			fbwritevaluetoword(iValue:=0, iStartBit:=0, iEndBit:=7, wDataWord:=awBusDataToVTEM[1], xError=> );							// Addressed Target = 0 (ignored)
			fbwritevaluetoword(iValue:=0, iStartBit:=8, iEndBit:=15, wDataWord:=awBusDataToVTEM[1], xError=> );							// Index = 0 (ignored)
			fbwritevaluetoword(iValue:=0, iStartBit:=0, iEndBit:=15, wDataWord:=awBusDataToVTEM[2], xError=> );							// Value = 0 (ignored)
			
		6:	// STOP RUNNING MOTION APP
			fbwritevaluetoword(iValue:=61, iStartBit:=0, iEndBit:=5, wDataWord:=awBusDataToVTEM[0], xError=> );							// Valve Mode = 61 (stop)
			fbwritevaluetoword(iValue:=0, iStartBit:=6, iEndBit:=7, wDataWord:=awBusDataToVTEM[0], xError=> );							// App Control = 0 (unused)
			fbwritevaluetoword(iValue:=0, iStartBit:=8, iEndBit:=15, wDataWord:=awBusDataToVTEM[0], xError=> );							// App Option = 0 (unused)
			fbwritevaluetoword(iValue:=0, iStartBit:=0, iEndBit:=15, wDataWord:=awBusDataToVTEM[1], xError=> );							// Setpoint Value 1 = 0 (unused)
			fbwritevaluetoword(iValue:=0, iStartBit:=0, iEndBit:=15, wDataWord:=awBusDataToVTEM[2], xError=> );							// Setpoint Value 2 = 0 (unused)
		
		30:	// RUN FB_UPLOADMULTIPLEPARAMETERS
			fbuploadMultipleParameters(
				awBusDataFromVTEM:= awBusDataFromVTEM, 
				awBusDataToVTEM:= awBusDataToVTEM, 
				xExecute:= TRUE, 
				iResponse=> , 
				iCurrentValue=> , 
				xUploadDone=> , 
				xUploadError=> , 
				aTransferPackages:= aTransferPackages);

		40:	// RESET FB_UPLOADMULTIPLEPARAMETERS
			fbuploadMultipleParameters(
				awBusDataFromVTEM:= awBusDataFromVTEM, 
				awBusDataToVTEM:= awBusDataToVTEM, 
				xExecute:= FALSE, 
				iResponse=> , 
				iCurrentValue=> , 
				xUploadDone=> , 
				xUploadError=> , 
				aTransferPackages:= aTransferPackages);
	END_CASE
//-----------------------------------------------------------------------------------------------------------

END_FUNCTION_BLOCK

// Transfermode/specific_MA_config/FB_Read_config_MA_03
/// This function block can be used to upload the configuration of Motion App 3 ("Proportional pressure regulation").
/// The specific parameters of this Motion App are the outputs of this FB
/// The function block uses the transfer mode to read this configuration from the Motion Terminal
/// and indicates the state of the upload process at the output iResponse.

FUNCTION_BLOCK FB_Read_config_MA_03
VAR_INPUT
	awBusDataFromVTEM 				: ARRAY [0..2] OF WORD;		// array of 3 words of process data received from the Motion Terminal
END_VAR
	
VAR_IN_OUT
	awBusDataToVTEM 				: ARRAY [0..2] OF WORD; 	// array of 3 words of process data sent to the Motion Terminal
END_VAR

VAR_INPUT
	xExecute 						: BOOL; 					// rising edge starts the reading process, falling edge resets the function block after reading is done
	xAbort							: BOOL;						// rising edge aborts the reading process
	iParameterSet					: INT := 1; 				// the parameter set to be read from, 1 by default
END_VAR                     		

VAR_OUTPUT                  		
	// system parameters
		iInPortRetracted_optional	: INT;						// Sensor port for detection of end position at pressurisation of outlet port 2 (retracted), value is number of the slot (beginning from 0 and including valve slots) * 10 + number of the port
		iInPortAdvanced_optional	: INT;						// Sensor port for detection of end position at pressurisation of outlet port 4 (advanced), value is number of the slot (beginning from 0 and including valve slots) * 10 + number of the port
		
	// application parameters
		iCharacteristicAt2 			: INT;		 				// characteristic of the control algorithm for outlet port 2 (0 = small volumes ≥0.05 l … ≤0.1 l, 1 = medium volumes >0.1 l … <1.0 l, 2 = large volumes ≥1.0 l, 3 = customized characteristic defined by tuning parameters)
		iCharacteristicAt4 			: INT; 						// characteristic of the control algorithm for outlet port 4 (0 = small volumes ≥0.05 l … ≤0.1 l, 1 = medium volumes >0.1 l … <1.0 l, 2 = large volumes ≥1.0 l, 3 = customized characteristic defined by tuning parameters)

	//tuning parameters
		iOptProportionalGainFor2	: INT;						// Optional tuning parameter for the customized proportional element of the PID modulator at outlet port 2 [1 digit = 0.01 g/s/bar]
		iOptIntegralGainFor2		: INT;						// Optional tuning parameter for the customized integral element of the PID modulator at outlet port 2 [1 digit = 0.01 g/s²/bar]
		iOptTimeConstantFor2		: INT;						// Optional tuning parameter for the customized time constant element of the PID modulator at outlet port 2 [1 digit = 0.001 s]
		iOptShiftZeroPointSwitchOff2	: INT;					// Optional tuning parameter for shifting the zero point switch-off for outlet port 2 [1 digit = 0.001 bar]
		iOptProportionalGainFor4	: INT;						// Optional tuning parameter for the customized proportional element of the PID modulator at outlet port 4 [1 digit = 0.01 g/s/bar]
		iOptIntegralGainFor4		: INT;						// Optional tuning parameter for the customized integral element of the PID modulator at outlet port 4 [1 digit = 0.01 g/s²/bar]
		iOptTimeConstantFor4		: INT;						// Optional tuning parameter for the customized time constant element of the PID modulator at outlet port 4 [1 digit = 0.001 s]
		iOptShiftZeroPointSwitchOff4	: INT;					// Optional tuning parameter for shifting the zero point switch-off for outlet port 4 [1 digit = 0.001 bar]
		
	// function block response
		iResponse 					: eTransferResponse; 		// returns the status of the upload process
		xBusy						: BOOL;						// TRUE as long as the upload process is running
		xDone 						: BOOL; 					// indicates whether the upload was successfull
		xError 						: BOOL; 					// indicates whether an error occurred during the transfer
		xAborted					: BOOL;						// TRUE if the function block was canceled by xAbort	
END_VAR

VAR
	iState							: INT := 10;
	xStateChange					: BOOL;
	iCommandNumber					: INT;
	xFirstCycle						: BOOL := TRUE;				// indicator for the first cycle of the function block
	iParameterSetFC					: INT;						// value on input iParameterSet during first cycle
	
	aTransferPackages				: ARRAY [0..100] OF stTransferPackage;
	fbreadbitsfromword				: FB_Read_Bits_From_Word;
	fbuploadMultipleParameters 		: FB_Upload_Multiple_Parameters;
	fbWriteValueToWord 				: FB_Write_Value_To_Word;

	iCounterResetArray				: INT;

	iCurrentValveMode				: INT;						//
END_VAR

(*****************************************************************************************************

Festo SE & Co. KG, Esslingen
Copyright (c) 2021. All rights reserved.

Product:            Motion Terminal VTEM
Description:        Function Block to upload the parameters for Motion App 3 from the Motion Terminal

Object version:     2.00
Last change:        2021-07
======================================================================================================
                                       H I S T O R Y
======================================================================================================
Version:            2.00
Date:               2021-07
Change/Activity:    - created (#3872357)
Release:            3.5.7.237 (CODESYS 3.5.7.2, Lib version 3.7)
Author:             JEBU
======================================================================================================

*****************************************************************************************************)

// pre-check of the value for the parameter set
	IF xExecute = TRUE AND (iParameterSet < 1 OR iParameterSet > 5) THEN		// invalid input for the parameter set
		xDone := FALSE; 
		xError := TRUE; 
		iResponse := eTransferResponse.invalid_ParameterSet;
		xStateChange := TRUE;
		iState := 70;	// ERROR
	END_IF
//-----------------------------------------------------------------------------------------------------------

// check if iParameterSet was changed
	IF xExecute = TRUE AND xFirstCycle = TRUE THEN
		xFirstCycle := FALSE;
		iParameterSetFC := iParameterSet;
	END_IF
	
	IF xExecute = TRUE AND iParameterSet <> iParameterSetFC THEN
		xStateChange := TRUE;
		iState := 70;
		iResponse := eTransferResponse.FB_needs_rising_edge_xExecute;
	END_IF
//-----------------------------------------------------------------------------------------------------------

// WRITE PARAMETER INDICES INTO ARRAY
	//iCharacteristicAt2
		aTransferPackages[0].iChannel := iParameterSet;
		aTransferPackages[0].iAddressedTarget := 3;
		aTransferPackages[0].iIndex := 220;
		
	//iCharacteristicAt4
		aTransferPackages[1].iChannel := iParameterSet;
		aTransferPackages[1].iAddressedTarget := 3;
		aTransferPackages[1].iIndex := 221;
		
	//iOptProportionalGainFor2
		aTransferPackages[2].iChannel := iParameterSet;
		aTransferPackages[2].iAddressedTarget := 3;
		aTransferPackages[2].iIndex := 230;
		
	//iOptIntegralGainFor2
		aTransferPackages[3].iChannel := iParameterSet;
		aTransferPackages[3].iAddressedTarget := 3;
		aTransferPackages[3].iIndex := 231;
		
	//iOptTimeConstantFor2
		aTransferPackages[4].iChannel := iParameterSet;
		aTransferPackages[4].iAddressedTarget := 3;
		aTransferPackages[4].iIndex := 232;
		
	//iOptShiftZeroPointSwitchOff2
		aTransferPackages[5].iChannel := iParameterSet;
		aTransferPackages[5].iAddressedTarget := 3;
		aTransferPackages[5].iIndex := 233;
		
	//iOptProportionalGainFor4
		aTransferPackages[6].iChannel := iParameterSet;
		aTransferPackages[6].iAddressedTarget := 3;
		aTransferPackages[6].iIndex := 240;
		
	//iOptIntegralGainFor4
		aTransferPackages[7].iChannel := iParameterSet;
		aTransferPackages[7].iAddressedTarget := 3;
		aTransferPackages[7].iIndex := 241;
		
	//iOptTimeConstantFor4
		aTransferPackages[8].iChannel := iParameterSet;
		aTransferPackages[8].iAddressedTarget := 3;
		aTransferPackages[8].iIndex := 242;
		
	//iOptShiftZeroPointSwitchOff4
		aTransferPackages[9].iChannel := iParameterSet;
		aTransferPackages[9].iAddressedTarget := 3;
		aTransferPackages[9].iIndex := 243;
		
	//iInPortRetract_optional
		aTransferPackages[10].iChannel := iParameterSet;
		aTransferPackages[10].iAddressedTarget := 3;
		aTransferPackages[10].iIndex := 70;
		
	//iInPortAdvanced_optional
		aTransferPackages[11].iChannel := iParameterSet;
		aTransferPackages[11].iAddressedTarget := 3;
		aTransferPackages[11].iIndex := 71;
		
	// define end of parameter list to be uploaded by setting all variables to 0 (end criterion for FB_Upload_Multiple_Parameters)
		aTransferPackages[12].iChannel := 0;
		aTransferPackages[12].iAddressedTarget := 0;
		aTransferPackages[12].iIndex := 0;
//-----------------------------------------------------------------------------------------------------------

// Read the current status of the the motion terminal
	fbreadbitsfromword(wData:= awBusDataFromVTEM[0], iStartBit:=0, iEndBit:= 5, iValue=> iCurrentValveMode, xError=> );				// read current valve mode
//-----------------------------------------------------------------------------------------------------------

// Transition: Aborting condition when xAbort is TRUE in all States except "IDLE" , "ABORTING" and "RESETTING"
	IF xAbort = TRUE AND NOT(iState = 10 AND xExecute = FALSE) AND iState <> 80 AND iState <> 100 THEN
		xStateChange := TRUE;	// Leaving current state
		iState := 80;	// Choosing next state, here: ABORTING
	END_IF
//-----------------------------------------------------------------------------------------------------------

// local state machine
	CASE iState OF
		10:	// IDLE
			// code that is executed only in the first cycle of this state
				IF xStateChange = TRUE THEN
					xStateChange := FALSE;
					iResponse := eTransferResponse.ready_for_new_transfer;
					xDone := FALSE;
					xError := FALSE;
					xBusy := FALSE;
					xAborted := FALSE;
				END_IF
			//-----------------------------------------------------------------------------------------------------------
			
			// code that is repeated every cycle in this state
				iCommandNumber := 0;
			//-----------------------------------------------------------------------------------------------------------
			
			// Transition
			IF xExecute = TRUE THEN
				xStateChange := TRUE;
				iState := 20;
			END_IF
			//-----------------------------------------------------------------------------------------------------------
		
		20:	// RESETTING VALVE MODE TO 61
			// code that is executed only in the first cycle of this state
				IF xStateChange = TRUE THEN
					xStateChange := FALSE;
					iResponse := eTransferResponse.preparing_transfer;
					xDone := FALSE;
					xError := FALSE;
					xBusy := TRUE;
					xAborted := FALSE;
				END_IF
			//-----------------------------------------------------------------------------------------------------------
			
			// code that is repeated every cycle in this state	
				IF iCurrentValveMode = 63 THEN
					iCommandNumber := 5;	// exit transfer mode
				ELSIF iCurrentValveMode <> 61 AND iCurrentValveMode <> 63 THEN
					iCommandNumber := 6;	// stop running motion apps
				END_IF 
			//-----------------------------------------------------------------------------------------------------------
			
			// Transition
				IF iCurrentValveMode = 61 THEN
					xStateChange := TRUE;	// Leave this state
					iState := 30;
					iCommandNumber := 30;			
				END_IF
			//-----------------------------------------------------------------------------------------------------------
		
		30:	// READING PARAMETER VALUES
			// code that is executed only in the first cycle of this state
				IF xStateChange = TRUE THEN
					xStateChange := FALSE;
					iResponse := eTransferResponse.transferring;
					xDone := FALSE;
					xError := FALSE;
					xBusy := TRUE;
					xAborted := FALSE;
				END_IF
			//-----------------------------------------------------------------------------------------------------------
			
			// code that is repeated every cycle in this state
				iCommandNumber := 30;		// read parameter values
			//-----------------------------------------------------------------------------------------------------------
			
			// Transition
				IF fbuploadMultipleParameters.xExecute = TRUE AND fbuploadMultipleParameters.xUploadDone = TRUE AND fbuploadMultipleParameters.xUploadError = FALSE THEN	// Upload Done
					xStateChange := TRUE;
					iState := 40;	// Write parameter values to outputs
				ELSIF fbuploadMultipleParameters.xExecute = TRUE AND fbuploadMultipleParameters.xUploadDone = FALSE AND fbuploadMultipleParameters.xUploadError = TRUE THEN	// Error during update
					xStateChange := TRUE;
					iState := 70;	// ERROR
					iResponse := fbuploadMultipleParameters.iResponse;
				END_IF
			//-----------------------------------------------------------------------------------------------------------
		
		40:	// WRITE PARAMETER VALUES TO OUTPUTS
			// code that is executed only in the first cycle of this state
				IF xStateChange = TRUE THEN
					xStateChange := FALSE;
					iResponse := eTransferResponse.transferring;
					xDone := FALSE;
					xError := FALSE;
					xBusy := TRUE;
					xAborted := FALSE;
				END_IF
			//-----------------------------------------------------------------------------------------------------------
			
